   // GBK_TO_UNICODE[27068] := 16#CFB8;
   // GBK_TO_UNICODE[27069] := 16#7EC6;
   // GBK_TO_UNICODE[27070] := 16#CFB9;
   // GBK_TO_UNICODE[27071] := 16#778E;
   // GBK_TO_UNICODE[27072] := 16#CFBA;
   // GBK_TO_UNICODE[27073] := 16#867E;
   // GBK_TO_UNICODE[27074] := 16#CFBB;
   // GBK_TO_UNICODE[27075] := 16#5323;
   // GBK_TO_UNICODE[27076] := 16#CFBC;
   // GBK_TO_UNICODE[27077] := 16#971E;
   // GBK_TO_UNICODE[27078] := 16#CFBD;
   // GBK_TO_UNICODE[27079] := 16#8F96;
   // GBK_TO_UNICODE[27080] := 16#CFBE;
   // GBK_TO_UNICODE[27081] := 16#6687;
   // GBK_TO_UNICODE[27082] := 16#CFBF;
   // GBK_TO_UNICODE[27083] := 16#5CE1;
   // GBK_TO_UNICODE[27084] := 16#CFC0;
   // GBK_TO_UNICODE[27085] := 16#4FA0;
   // GBK_TO_UNICODE[27086] := 16#CFC1;
   // GBK_TO_UNICODE[27087] := 16#72ED;
   // GBK_TO_UNICODE[27088] := 16#CFC2;
   // GBK_TO_UNICODE[27089] := 16#4E0B;
   // GBK_TO_UNICODE[27090] := 16#CFC3;
   // GBK_TO_UNICODE[27091] := 16#53A6;
   // GBK_TO_UNICODE[27092] := 16#CFC4;
   // GBK_TO_UNICODE[27093] := 16#590F;
   // GBK_TO_UNICODE[27094] := 16#CFC5;
   // GBK_TO_UNICODE[27095] := 16#5413;
   // GBK_TO_UNICODE[27096] := 16#CFC6;
   // GBK_TO_UNICODE[27097] := 16#6380;
   // GBK_TO_UNICODE[27098] := 16#CFC7;
   // GBK_TO_UNICODE[27099] := 16#9528;
   // GBK_TO_UNICODE[27100] := 16#CFC8;
   // GBK_TO_UNICODE[27101] := 16#5148;
   // GBK_TO_UNICODE[27102] := 16#CFC9;
   // GBK_TO_UNICODE[27103] := 16#4ED9;
   // GBK_TO_UNICODE[27104] := 16#CFCA;
   // GBK_TO_UNICODE[27105] := 16#9C9C;
   // GBK_TO_UNICODE[27106] := 16#CFCB;
   // GBK_TO_UNICODE[27107] := 16#7EA4;
   // GBK_TO_UNICODE[27108] := 16#CFCC;
   // GBK_TO_UNICODE[27109] := 16#54B8;
   // GBK_TO_UNICODE[27110] := 16#CFCD;
   // GBK_TO_UNICODE[27111] := 16#8D24;
   // GBK_TO_UNICODE[27112] := 16#CFCE;
   // GBK_TO_UNICODE[27113] := 16#8854;
   // GBK_TO_UNICODE[27114] := 16#CFCF;
   // GBK_TO_UNICODE[27115] := 16#8237;
   // GBK_TO_UNICODE[27116] := 16#CFD0;
   // GBK_TO_UNICODE[27117] := 16#95F2;
   // GBK_TO_UNICODE[27118] := 16#CFD1;
   // GBK_TO_UNICODE[27119] := 16#6D8E;
   // GBK_TO_UNICODE[27120] := 16#CFD2;
   // GBK_TO_UNICODE[27121] := 16#5F26;
   // GBK_TO_UNICODE[27122] := 16#CFD3;
   // GBK_TO_UNICODE[27123] := 16#5ACC;
   // GBK_TO_UNICODE[27124] := 16#CFD4;
   // GBK_TO_UNICODE[27125] := 16#663E;
   // GBK_TO_UNICODE[27126] := 16#CFD5;
   // GBK_TO_UNICODE[27127] := 16#9669;
   // GBK_TO_UNICODE[27128] := 16#CFD6;
   // GBK_TO_UNICODE[27129] := 16#73B0;
   // GBK_TO_UNICODE[27130] := 16#CFD7;
   // GBK_TO_UNICODE[27131] := 16#732E;
   // GBK_TO_UNICODE[27132] := 16#CFD8;
   // GBK_TO_UNICODE[27133] := 16#53BF;
   // GBK_TO_UNICODE[27134] := 16#CFD9;
   // GBK_TO_UNICODE[27135] := 16#817A;
   // GBK_TO_UNICODE[27136] := 16#CFDA;
   // GBK_TO_UNICODE[27137] := 16#9985;
   // GBK_TO_UNICODE[27138] := 16#CFDB;
   // GBK_TO_UNICODE[27139] := 16#7FA1;
   // GBK_TO_UNICODE[27140] := 16#CFDC;
   // GBK_TO_UNICODE[27141] := 16#5BAA;
   // GBK_TO_UNICODE[27142] := 16#CFDD;
   // GBK_TO_UNICODE[27143] := 16#9677;
   // GBK_TO_UNICODE[27144] := 16#CFDE;
   // GBK_TO_UNICODE[27145] := 16#9650;
   // GBK_TO_UNICODE[27146] := 16#CFDF;
   // GBK_TO_UNICODE[27147] := 16#7EBF;
   // GBK_TO_UNICODE[27148] := 16#CFE0;
   // GBK_TO_UNICODE[27149] := 16#76F8;
   // GBK_TO_UNICODE[27150] := 16#CFE1;
   // GBK_TO_UNICODE[27151] := 16#53A2;
   // GBK_TO_UNICODE[27152] := 16#CFE2;
   // GBK_TO_UNICODE[27153] := 16#9576;
   // GBK_TO_UNICODE[27154] := 16#CFE3;
   // GBK_TO_UNICODE[27155] := 16#9999;
   // GBK_TO_UNICODE[27156] := 16#CFE4;
   // GBK_TO_UNICODE[27157] := 16#7BB1;
   // GBK_TO_UNICODE[27158] := 16#CFE5;
   // GBK_TO_UNICODE[27159] := 16#8944;
   // GBK_TO_UNICODE[27160] := 16#CFE6;
   // GBK_TO_UNICODE[27161] := 16#6E58;
   // GBK_TO_UNICODE[27162] := 16#CFE7;
   // GBK_TO_UNICODE[27163] := 16#4E61;
   // GBK_TO_UNICODE[27164] := 16#CFE8;
   // GBK_TO_UNICODE[27165] := 16#7FD4;
   // GBK_TO_UNICODE[27166] := 16#CFE9;
   // GBK_TO_UNICODE[27167] := 16#7965;
   // GBK_TO_UNICODE[27168] := 16#CFEA;
   // GBK_TO_UNICODE[27169] := 16#8BE6;
   // GBK_TO_UNICODE[27170] := 16#CFEB;
   // GBK_TO_UNICODE[27171] := 16#60F3;
   // GBK_TO_UNICODE[27172] := 16#CFEC;
   // GBK_TO_UNICODE[27173] := 16#54CD;
   // GBK_TO_UNICODE[27174] := 16#CFED;
   // GBK_TO_UNICODE[27175] := 16#4EAB;
   // GBK_TO_UNICODE[27176] := 16#CFEE;
   // GBK_TO_UNICODE[27177] := 16#9879;
   // GBK_TO_UNICODE[27178] := 16#CFEF;
   // GBK_TO_UNICODE[27179] := 16#5DF7;
   // GBK_TO_UNICODE[27180] := 16#CFF0;
   // GBK_TO_UNICODE[27181] := 16#6A61;
   // GBK_TO_UNICODE[27182] := 16#CFF1;
   // GBK_TO_UNICODE[27183] := 16#50CF;
   // GBK_TO_UNICODE[27184] := 16#CFF2;
   // GBK_TO_UNICODE[27185] := 16#5411;
   // GBK_TO_UNICODE[27186] := 16#CFF3;
   // GBK_TO_UNICODE[27187] := 16#8C61;
   // GBK_TO_UNICODE[27188] := 16#CFF4;
   // GBK_TO_UNICODE[27189] := 16#8427;
   // GBK_TO_UNICODE[27190] := 16#CFF5;
   // GBK_TO_UNICODE[27191] := 16#785D;
   // GBK_TO_UNICODE[27192] := 16#CFF6;
   // GBK_TO_UNICODE[27193] := 16#9704;
   // GBK_TO_UNICODE[27194] := 16#CFF7;
   // GBK_TO_UNICODE[27195] := 16#524A;
   // GBK_TO_UNICODE[27196] := 16#CFF8;
   // GBK_TO_UNICODE[27197] := 16#54EE;
   // GBK_TO_UNICODE[27198] := 16#CFF9;
   // GBK_TO_UNICODE[27199] := 16#56A3;
   // GBK_TO_UNICODE[27200] := 16#CFFA;
   // GBK_TO_UNICODE[27201] := 16#9500;
   // GBK_TO_UNICODE[27202] := 16#CFFB;
   // GBK_TO_UNICODE[27203] := 16#6D88;
   // GBK_TO_UNICODE[27204] := 16#CFFC;
   // GBK_TO_UNICODE[27205] := 16#5BB5;
   // GBK_TO_UNICODE[27206] := 16#CFFD;
   // GBK_TO_UNICODE[27207] := 16#6DC6;
   // GBK_TO_UNICODE[27208] := 16#CFFE;
   // GBK_TO_UNICODE[27209] := 16#6653;
   // GBK_TO_UNICODE[27210] := 16#D040;
   // GBK_TO_UNICODE[27211] := 16#8824;
   // GBK_TO_UNICODE[27212] := 16#D041;
   // GBK_TO_UNICODE[27213] := 16#8825;
   // GBK_TO_UNICODE[27214] := 16#D042;
   // GBK_TO_UNICODE[27215] := 16#8826;
   // GBK_TO_UNICODE[27216] := 16#D043;
   // GBK_TO_UNICODE[27217] := 16#8827;
   // GBK_TO_UNICODE[27218] := 16#D044;
   // GBK_TO_UNICODE[27219] := 16#8828;
   // GBK_TO_UNICODE[27220] := 16#D045;
   // GBK_TO_UNICODE[27221] := 16#8829;
   // GBK_TO_UNICODE[27222] := 16#D046;
   // GBK_TO_UNICODE[27223] := 16#882A;
   // GBK_TO_UNICODE[27224] := 16#D047;
   // GBK_TO_UNICODE[27225] := 16#882B;
   // GBK_TO_UNICODE[27226] := 16#D048;
   // GBK_TO_UNICODE[27227] := 16#882C;
   // GBK_TO_UNICODE[27228] := 16#D049;
   // GBK_TO_UNICODE[27229] := 16#882D;
   // GBK_TO_UNICODE[27230] := 16#D04A;
   // GBK_TO_UNICODE[27231] := 16#882E;
   // GBK_TO_UNICODE[27232] := 16#D04B;
   // GBK_TO_UNICODE[27233] := 16#882F;
   // GBK_TO_UNICODE[27234] := 16#D04C;
   // GBK_TO_UNICODE[27235] := 16#8830;
   // GBK_TO_UNICODE[27236] := 16#D04D;
   // GBK_TO_UNICODE[27237] := 16#8831;
   // GBK_TO_UNICODE[27238] := 16#D04E;
   // GBK_TO_UNICODE[27239] := 16#8833;
   // GBK_TO_UNICODE[27240] := 16#D04F;
   // GBK_TO_UNICODE[27241] := 16#8834;
   // GBK_TO_UNICODE[27242] := 16#D050;
   // GBK_TO_UNICODE[27243] := 16#8835;
   // GBK_TO_UNICODE[27244] := 16#D051;
   // GBK_TO_UNICODE[27245] := 16#8836;
   // GBK_TO_UNICODE[27246] := 16#D052;
   // GBK_TO_UNICODE[27247] := 16#8837;
   // GBK_TO_UNICODE[27248] := 16#D053;
   // GBK_TO_UNICODE[27249] := 16#8838;
   // GBK_TO_UNICODE[27250] := 16#D054;
   // GBK_TO_UNICODE[27251] := 16#883A;
   // GBK_TO_UNICODE[27252] := 16#D055;
   // GBK_TO_UNICODE[27253] := 16#883B;
   // GBK_TO_UNICODE[27254] := 16#D056;
   // GBK_TO_UNICODE[27255] := 16#883D;
   // GBK_TO_UNICODE[27256] := 16#D057;
   // GBK_TO_UNICODE[27257] := 16#883E;
   // GBK_TO_UNICODE[27258] := 16#D058;
   // GBK_TO_UNICODE[27259] := 16#883F;
   // GBK_TO_UNICODE[27260] := 16#D059;
   // GBK_TO_UNICODE[27261] := 16#8841;
   // GBK_TO_UNICODE[27262] := 16#D05A;
   // GBK_TO_UNICODE[27263] := 16#8842;
   // GBK_TO_UNICODE[27264] := 16#D05B;
   // GBK_TO_UNICODE[27265] := 16#8843;
   // GBK_TO_UNICODE[27266] := 16#D05C;
   // GBK_TO_UNICODE[27267] := 16#8846;
   // GBK_TO_UNICODE[27268] := 16#D05D;
   // GBK_TO_UNICODE[27269] := 16#8847;
   // GBK_TO_UNICODE[27270] := 16#D05E;
   // GBK_TO_UNICODE[27271] := 16#8848;
   // GBK_TO_UNICODE[27272] := 16#D05F;
   // GBK_TO_UNICODE[27273] := 16#8849;
   // GBK_TO_UNICODE[27274] := 16#D060;
   // GBK_TO_UNICODE[27275] := 16#884A;
   // GBK_TO_UNICODE[27276] := 16#D061;
   // GBK_TO_UNICODE[27277] := 16#884B;
   // GBK_TO_UNICODE[27278] := 16#D062;
   // GBK_TO_UNICODE[27279] := 16#884E;
   // GBK_TO_UNICODE[27280] := 16#D063;
   // GBK_TO_UNICODE[27281] := 16#884F;
   // GBK_TO_UNICODE[27282] := 16#D064;
   // GBK_TO_UNICODE[27283] := 16#8850;
   // GBK_TO_UNICODE[27284] := 16#D065;
   // GBK_TO_UNICODE[27285] := 16#8851;
   // GBK_TO_UNICODE[27286] := 16#D066;
   // GBK_TO_UNICODE[27287] := 16#8852;
   // GBK_TO_UNICODE[27288] := 16#D067;
   // GBK_TO_UNICODE[27289] := 16#8853;
   // GBK_TO_UNICODE[27290] := 16#D068;
   // GBK_TO_UNICODE[27291] := 16#8855;
   // GBK_TO_UNICODE[27292] := 16#D069;
   // GBK_TO_UNICODE[27293] := 16#8856;
   // GBK_TO_UNICODE[27294] := 16#D06A;
   // GBK_TO_UNICODE[27295] := 16#8858;
   // GBK_TO_UNICODE[27296] := 16#D06B;
   // GBK_TO_UNICODE[27297] := 16#885A;
   // GBK_TO_UNICODE[27298] := 16#D06C;
   // GBK_TO_UNICODE[27299] := 16#885B;
   // GBK_TO_UNICODE[27300] := 16#D06D;
   // GBK_TO_UNICODE[27301] := 16#885C;
   // GBK_TO_UNICODE[27302] := 16#D06E;
   // GBK_TO_UNICODE[27303] := 16#885D;
   // GBK_TO_UNICODE[27304] := 16#D06F;
   // GBK_TO_UNICODE[27305] := 16#885E;
   // GBK_TO_UNICODE[27306] := 16#D070;
   // GBK_TO_UNICODE[27307] := 16#885F;
   // GBK_TO_UNICODE[27308] := 16#D071;
   // GBK_TO_UNICODE[27309] := 16#8860;
   // GBK_TO_UNICODE[27310] := 16#D072;
   // GBK_TO_UNICODE[27311] := 16#8866;
   // GBK_TO_UNICODE[27312] := 16#D073;
   // GBK_TO_UNICODE[27313] := 16#8867;
   // GBK_TO_UNICODE[27314] := 16#D074;
   // GBK_TO_UNICODE[27315] := 16#886A;
   // GBK_TO_UNICODE[27316] := 16#D075;
   // GBK_TO_UNICODE[27317] := 16#886D;
   // GBK_TO_UNICODE[27318] := 16#D076;
   // GBK_TO_UNICODE[27319] := 16#886F;
   // GBK_TO_UNICODE[27320] := 16#D077;
   // GBK_TO_UNICODE[27321] := 16#8871;
   // GBK_TO_UNICODE[27322] := 16#D078;
   // GBK_TO_UNICODE[27323] := 16#8873;
   // GBK_TO_UNICODE[27324] := 16#D079;
   // GBK_TO_UNICODE[27325] := 16#8874;
   // GBK_TO_UNICODE[27326] := 16#D07A;
   // GBK_TO_UNICODE[27327] := 16#8875;
   // GBK_TO_UNICODE[27328] := 16#D07B;
   // GBK_TO_UNICODE[27329] := 16#8876;
   // GBK_TO_UNICODE[27330] := 16#D07C;
   // GBK_TO_UNICODE[27331] := 16#8878;
   // GBK_TO_UNICODE[27332] := 16#D07D;
   // GBK_TO_UNICODE[27333] := 16#8879;
   // GBK_TO_UNICODE[27334] := 16#D07E;
   // GBK_TO_UNICODE[27335] := 16#887A;
   // GBK_TO_UNICODE[27336] := 16#D080;
   // GBK_TO_UNICODE[27337] := 16#887B;
   // GBK_TO_UNICODE[27338] := 16#D081;
   // GBK_TO_UNICODE[27339] := 16#887C;
   // GBK_TO_UNICODE[27340] := 16#D082;
   // GBK_TO_UNICODE[27341] := 16#8880;
   // GBK_TO_UNICODE[27342] := 16#D083;
   // GBK_TO_UNICODE[27343] := 16#8883;
   // GBK_TO_UNICODE[27344] := 16#D084;
   // GBK_TO_UNICODE[27345] := 16#8886;
   // GBK_TO_UNICODE[27346] := 16#D085;
   // GBK_TO_UNICODE[27347] := 16#8887;
   // GBK_TO_UNICODE[27348] := 16#D086;
   // GBK_TO_UNICODE[27349] := 16#8889;
   // GBK_TO_UNICODE[27350] := 16#D087;
   // GBK_TO_UNICODE[27351] := 16#888A;
   // GBK_TO_UNICODE[27352] := 16#D088;
   // GBK_TO_UNICODE[27353] := 16#888C;
   // GBK_TO_UNICODE[27354] := 16#D089;
   // GBK_TO_UNICODE[27355] := 16#888E;
   // GBK_TO_UNICODE[27356] := 16#D08A;
   // GBK_TO_UNICODE[27357] := 16#888F;
   // GBK_TO_UNICODE[27358] := 16#D08B;
   // GBK_TO_UNICODE[27359] := 16#8890;
   // GBK_TO_UNICODE[27360] := 16#D08C;
   // GBK_TO_UNICODE[27361] := 16#8891;
   // GBK_TO_UNICODE[27362] := 16#D08D;
   // GBK_TO_UNICODE[27363] := 16#8893;
   // GBK_TO_UNICODE[27364] := 16#D08E;
   // GBK_TO_UNICODE[27365] := 16#8894;
   // GBK_TO_UNICODE[27366] := 16#D08F;
   // GBK_TO_UNICODE[27367] := 16#8895;
   // GBK_TO_UNICODE[27368] := 16#D090;
   // GBK_TO_UNICODE[27369] := 16#8897;
   // GBK_TO_UNICODE[27370] := 16#D091;
   // GBK_TO_UNICODE[27371] := 16#8898;
   // GBK_TO_UNICODE[27372] := 16#D092;
   // GBK_TO_UNICODE[27373] := 16#8899;
   // GBK_TO_UNICODE[27374] := 16#D093;
   // GBK_TO_UNICODE[27375] := 16#889A;
   // GBK_TO_UNICODE[27376] := 16#D094;
   // GBK_TO_UNICODE[27377] := 16#889B;
   // GBK_TO_UNICODE[27378] := 16#D095;
   // GBK_TO_UNICODE[27379] := 16#889D;
   // GBK_TO_UNICODE[27380] := 16#D096;
   // GBK_TO_UNICODE[27381] := 16#889E;
   // GBK_TO_UNICODE[27382] := 16#D097;
   // GBK_TO_UNICODE[27383] := 16#889F;
   // GBK_TO_UNICODE[27384] := 16#D098;
   // GBK_TO_UNICODE[27385] := 16#88A0;
   // GBK_TO_UNICODE[27386] := 16#D099;
   // GBK_TO_UNICODE[27387] := 16#88A1;
   // GBK_TO_UNICODE[27388] := 16#D09A;
   // GBK_TO_UNICODE[27389] := 16#88A3;
   // GBK_TO_UNICODE[27390] := 16#D09B;
   // GBK_TO_UNICODE[27391] := 16#88A5;
   // GBK_TO_UNICODE[27392] := 16#D09C;
   // GBK_TO_UNICODE[27393] := 16#88A6;
   // GBK_TO_UNICODE[27394] := 16#D09D;
   // GBK_TO_UNICODE[27395] := 16#88A7;
   // GBK_TO_UNICODE[27396] := 16#D09E;
   // GBK_TO_UNICODE[27397] := 16#88A8;
   // GBK_TO_UNICODE[27398] := 16#D09F;
   // GBK_TO_UNICODE[27399] := 16#88A9;
   // GBK_TO_UNICODE[27400] := 16#D0A0;
   // GBK_TO_UNICODE[27401] := 16#88AA;
   // GBK_TO_UNICODE[27402] := 16#D0A1;
   // GBK_TO_UNICODE[27403] := 16#5C0F;
   // GBK_TO_UNICODE[27404] := 16#D0A2;
   // GBK_TO_UNICODE[27405] := 16#5B5D;
   // GBK_TO_UNICODE[27406] := 16#D0A3;
   // GBK_TO_UNICODE[27407] := 16#6821;
   // GBK_TO_UNICODE[27408] := 16#D0A4;
   // GBK_TO_UNICODE[27409] := 16#8096;
   // GBK_TO_UNICODE[27410] := 16#D0A5;
   // GBK_TO_UNICODE[27411] := 16#5578;
   // GBK_TO_UNICODE[27412] := 16#D0A6;
   // GBK_TO_UNICODE[27413] := 16#7B11;
   // GBK_TO_UNICODE[27414] := 16#D0A7;
   // GBK_TO_UNICODE[27415] := 16#6548;
   // GBK_TO_UNICODE[27416] := 16#D0A8;
   // GBK_TO_UNICODE[27417] := 16#6954;
   // GBK_TO_UNICODE[27418] := 16#D0A9;
   // GBK_TO_UNICODE[27419] := 16#4E9B;
   // GBK_TO_UNICODE[27420] := 16#D0AA;
   // GBK_TO_UNICODE[27421] := 16#6B47;
   // GBK_TO_UNICODE[27422] := 16#D0AB;
   // GBK_TO_UNICODE[27423] := 16#874E;
   // GBK_TO_UNICODE[27424] := 16#D0AC;
   // GBK_TO_UNICODE[27425] := 16#978B;
   // GBK_TO_UNICODE[27426] := 16#D0AD;
   // GBK_TO_UNICODE[27427] := 16#534F;
   // GBK_TO_UNICODE[27428] := 16#D0AE;
   // GBK_TO_UNICODE[27429] := 16#631F;
   // GBK_TO_UNICODE[27430] := 16#D0AF;
   // GBK_TO_UNICODE[27431] := 16#643A;
   // GBK_TO_UNICODE[27432] := 16#D0B0;
   // GBK_TO_UNICODE[27433] := 16#90AA;
   // GBK_TO_UNICODE[27434] := 16#D0B1;
   // GBK_TO_UNICODE[27435] := 16#659C;
   // GBK_TO_UNICODE[27436] := 16#D0B2;
   // GBK_TO_UNICODE[27437] := 16#80C1;
   // GBK_TO_UNICODE[27438] := 16#D0B3;
   // GBK_TO_UNICODE[27439] := 16#8C10;
   // GBK_TO_UNICODE[27440] := 16#D0B4;
   // GBK_TO_UNICODE[27441] := 16#5199;
   // GBK_TO_UNICODE[27442] := 16#D0B5;
   // GBK_TO_UNICODE[27443] := 16#68B0;
   // GBK_TO_UNICODE[27444] := 16#D0B6;
   // GBK_TO_UNICODE[27445] := 16#5378;
   // GBK_TO_UNICODE[27446] := 16#D0B7;
   // GBK_TO_UNICODE[27447] := 16#87F9;
   // GBK_TO_UNICODE[27448] := 16#D0B8;
   // GBK_TO_UNICODE[27449] := 16#61C8;
   // GBK_TO_UNICODE[27450] := 16#D0B9;
   // GBK_TO_UNICODE[27451] := 16#6CC4;
   // GBK_TO_UNICODE[27452] := 16#D0BA;
   // GBK_TO_UNICODE[27453] := 16#6CFB;
   // GBK_TO_UNICODE[27454] := 16#D0BB;
   // GBK_TO_UNICODE[27455] := 16#8C22;
   // GBK_TO_UNICODE[27456] := 16#D0BC;
   // GBK_TO_UNICODE[27457] := 16#5C51;
   // GBK_TO_UNICODE[27458] := 16#D0BD;
   // GBK_TO_UNICODE[27459] := 16#85AA;
   // GBK_TO_UNICODE[27460] := 16#D0BE;
   // GBK_TO_UNICODE[27461] := 16#82AF;
   // GBK_TO_UNICODE[27462] := 16#D0BF;
   // GBK_TO_UNICODE[27463] := 16#950C;
   // GBK_TO_UNICODE[27464] := 16#D0C0;
   // GBK_TO_UNICODE[27465] := 16#6B23;
   // GBK_TO_UNICODE[27466] := 16#D0C1;
   // GBK_TO_UNICODE[27467] := 16#8F9B;
   // GBK_TO_UNICODE[27468] := 16#D0C2;
   // GBK_TO_UNICODE[27469] := 16#65B0;
   // GBK_TO_UNICODE[27470] := 16#D0C3;
   // GBK_TO_UNICODE[27471] := 16#5FFB;
   // GBK_TO_UNICODE[27472] := 16#D0C4;
   // GBK_TO_UNICODE[27473] := 16#5FC3;
   // GBK_TO_UNICODE[27474] := 16#D0C5;
   // GBK_TO_UNICODE[27475] := 16#4FE1;
   // GBK_TO_UNICODE[27476] := 16#D0C6;
   // GBK_TO_UNICODE[27477] := 16#8845;
   // GBK_TO_UNICODE[27478] := 16#D0C7;
   // GBK_TO_UNICODE[27479] := 16#661F;
   // GBK_TO_UNICODE[27480] := 16#D0C8;
   // GBK_TO_UNICODE[27481] := 16#8165;
   // GBK_TO_UNICODE[27482] := 16#D0C9;
   // GBK_TO_UNICODE[27483] := 16#7329;
   // GBK_TO_UNICODE[27484] := 16#D0CA;
   // GBK_TO_UNICODE[27485] := 16#60FA;
   // GBK_TO_UNICODE[27486] := 16#D0CB;
   // GBK_TO_UNICODE[27487] := 16#5174;
   // GBK_TO_UNICODE[27488] := 16#D0CC;
   // GBK_TO_UNICODE[27489] := 16#5211;
   // GBK_TO_UNICODE[27490] := 16#D0CD;
   // GBK_TO_UNICODE[27491] := 16#578B;
   // GBK_TO_UNICODE[27492] := 16#D0CE;
   // GBK_TO_UNICODE[27493] := 16#5F62;
   // GBK_TO_UNICODE[27494] := 16#D0CF;
   // GBK_TO_UNICODE[27495] := 16#90A2;
   // GBK_TO_UNICODE[27496] := 16#D0D0;
   // GBK_TO_UNICODE[27497] := 16#884C;
   // GBK_TO_UNICODE[27498] := 16#D0D1;
   // GBK_TO_UNICODE[27499] := 16#9192;
   // GBK_TO_UNICODE[27500] := 16#D0D2;
   // GBK_TO_UNICODE[27501] := 16#5E78;
   // GBK_TO_UNICODE[27502] := 16#D0D3;
   // GBK_TO_UNICODE[27503] := 16#674F;
   // GBK_TO_UNICODE[27504] := 16#D0D4;
   // GBK_TO_UNICODE[27505] := 16#6027;
   // GBK_TO_UNICODE[27506] := 16#D0D5;
   // GBK_TO_UNICODE[27507] := 16#59D3;
   // GBK_TO_UNICODE[27508] := 16#D0D6;
   // GBK_TO_UNICODE[27509] := 16#5144;
   // GBK_TO_UNICODE[27510] := 16#D0D7;
   // GBK_TO_UNICODE[27511] := 16#51F6;
   // GBK_TO_UNICODE[27512] := 16#D0D8;
   // GBK_TO_UNICODE[27513] := 16#80F8;
   // GBK_TO_UNICODE[27514] := 16#D0D9;
   // GBK_TO_UNICODE[27515] := 16#5308;
   // GBK_TO_UNICODE[27516] := 16#D0DA;
   // GBK_TO_UNICODE[27517] := 16#6C79;
   // GBK_TO_UNICODE[27518] := 16#D0DB;
   // GBK_TO_UNICODE[27519] := 16#96C4;
   // GBK_TO_UNICODE[27520] := 16#D0DC;
   // GBK_TO_UNICODE[27521] := 16#718A;
   // GBK_TO_UNICODE[27522] := 16#D0DD;
   // GBK_TO_UNICODE[27523] := 16#4F11;
   // GBK_TO_UNICODE[27524] := 16#D0DE;
   // GBK_TO_UNICODE[27525] := 16#4FEE;
   // GBK_TO_UNICODE[27526] := 16#D0DF;
   // GBK_TO_UNICODE[27527] := 16#7F9E;
   // GBK_TO_UNICODE[27528] := 16#D0E0;
   // GBK_TO_UNICODE[27529] := 16#673D;
   // GBK_TO_UNICODE[27530] := 16#D0E1;
   // GBK_TO_UNICODE[27531] := 16#55C5;
   // GBK_TO_UNICODE[27532] := 16#D0E2;
   // GBK_TO_UNICODE[27533] := 16#9508;
   // GBK_TO_UNICODE[27534] := 16#D0E3;
   // GBK_TO_UNICODE[27535] := 16#79C0;
   // GBK_TO_UNICODE[27536] := 16#D0E4;
   // GBK_TO_UNICODE[27537] := 16#8896;
   // GBK_TO_UNICODE[27538] := 16#D0E5;
   // GBK_TO_UNICODE[27539] := 16#7EE3;
   // GBK_TO_UNICODE[27540] := 16#D0E6;
   // GBK_TO_UNICODE[27541] := 16#589F;
   // GBK_TO_UNICODE[27542] := 16#D0E7;
   // GBK_TO_UNICODE[27543] := 16#620C;
   // GBK_TO_UNICODE[27544] := 16#D0E8;
   // GBK_TO_UNICODE[27545] := 16#9700;
   // GBK_TO_UNICODE[27546] := 16#D0E9;
   // GBK_TO_UNICODE[27547] := 16#865A;
   // GBK_TO_UNICODE[27548] := 16#D0EA;
   // GBK_TO_UNICODE[27549] := 16#5618;
   // GBK_TO_UNICODE[27550] := 16#D0EB;
   // GBK_TO_UNICODE[27551] := 16#987B;
   // GBK_TO_UNICODE[27552] := 16#D0EC;
   // GBK_TO_UNICODE[27553] := 16#5F90;
   // GBK_TO_UNICODE[27554] := 16#D0ED;
   // GBK_TO_UNICODE[27555] := 16#8BB8;
   // GBK_TO_UNICODE[27556] := 16#D0EE;
   // GBK_TO_UNICODE[27557] := 16#84C4;
   // GBK_TO_UNICODE[27558] := 16#D0EF;
   // GBK_TO_UNICODE[27559] := 16#9157;
   // GBK_TO_UNICODE[27560] := 16#D0F0;
   // GBK_TO_UNICODE[27561] := 16#53D9;
   // GBK_TO_UNICODE[27562] := 16#D0F1;
   // GBK_TO_UNICODE[27563] := 16#65ED;
   // GBK_TO_UNICODE[27564] := 16#D0F2;
   // GBK_TO_UNICODE[27565] := 16#5E8F;
   // GBK_TO_UNICODE[27566] := 16#D0F3;
   // GBK_TO_UNICODE[27567] := 16#755C;
   // GBK_TO_UNICODE[27568] := 16#D0F4;
   // GBK_TO_UNICODE[27569] := 16#6064;
   // GBK_TO_UNICODE[27570] := 16#D0F5;
   // GBK_TO_UNICODE[27571] := 16#7D6E;
   // GBK_TO_UNICODE[27572] := 16#D0F6;
   // GBK_TO_UNICODE[27573] := 16#5A7F;
   // GBK_TO_UNICODE[27574] := 16#D0F7;
   // GBK_TO_UNICODE[27575] := 16#7EEA;
   // GBK_TO_UNICODE[27576] := 16#D0F8;
   // GBK_TO_UNICODE[27577] := 16#7EED;
   // GBK_TO_UNICODE[27578] := 16#D0F9;
   // GBK_TO_UNICODE[27579] := 16#8F69;
   // GBK_TO_UNICODE[27580] := 16#D0FA;
   // GBK_TO_UNICODE[27581] := 16#55A7;
   // GBK_TO_UNICODE[27582] := 16#D0FB;
   // GBK_TO_UNICODE[27583] := 16#5BA3;
   // GBK_TO_UNICODE[27584] := 16#D0FC;
   // GBK_TO_UNICODE[27585] := 16#60AC;
   // GBK_TO_UNICODE[27586] := 16#D0FD;
   // GBK_TO_UNICODE[27587] := 16#65CB;
   // GBK_TO_UNICODE[27588] := 16#D0FE;
   // GBK_TO_UNICODE[27589] := 16#7384;
   // GBK_TO_UNICODE[27590] := 16#D140;
   // GBK_TO_UNICODE[27591] := 16#88AC;
   // GBK_TO_UNICODE[27592] := 16#D141;
   // GBK_TO_UNICODE[27593] := 16#88AE;
   // GBK_TO_UNICODE[27594] := 16#D142;
   // GBK_TO_UNICODE[27595] := 16#88AF;
   // GBK_TO_UNICODE[27596] := 16#D143;
   // GBK_TO_UNICODE[27597] := 16#88B0;
   // GBK_TO_UNICODE[27598] := 16#D144;
   // GBK_TO_UNICODE[27599] := 16#88B2;
   // GBK_TO_UNICODE[27600] := 16#D145;
   // GBK_TO_UNICODE[27601] := 16#88B3;
   // GBK_TO_UNICODE[27602] := 16#D146;
   // GBK_TO_UNICODE[27603] := 16#88B4;
   // GBK_TO_UNICODE[27604] := 16#D147;
   // GBK_TO_UNICODE[27605] := 16#88B5;
   // GBK_TO_UNICODE[27606] := 16#D148;
   // GBK_TO_UNICODE[27607] := 16#88B6;
   // GBK_TO_UNICODE[27608] := 16#D149;
   // GBK_TO_UNICODE[27609] := 16#88B8;
   // GBK_TO_UNICODE[27610] := 16#D14A;
   // GBK_TO_UNICODE[27611] := 16#88B9;
   // GBK_TO_UNICODE[27612] := 16#D14B;
   // GBK_TO_UNICODE[27613] := 16#88BA;
   // GBK_TO_UNICODE[27614] := 16#D14C;
   // GBK_TO_UNICODE[27615] := 16#88BB;
   // GBK_TO_UNICODE[27616] := 16#D14D;
   // GBK_TO_UNICODE[27617] := 16#88BD;
   // GBK_TO_UNICODE[27618] := 16#D14E;
   // GBK_TO_UNICODE[27619] := 16#88BE;
   // GBK_TO_UNICODE[27620] := 16#D14F;
   // GBK_TO_UNICODE[27621] := 16#88BF;
   // GBK_TO_UNICODE[27622] := 16#D150;
   // GBK_TO_UNICODE[27623] := 16#88C0;
   // GBK_TO_UNICODE[27624] := 16#D151;
   // GBK_TO_UNICODE[27625] := 16#88C3;
   // GBK_TO_UNICODE[27626] := 16#D152;
   // GBK_TO_UNICODE[27627] := 16#88C4;
   // GBK_TO_UNICODE[27628] := 16#D153;
   // GBK_TO_UNICODE[27629] := 16#88C7;
   // GBK_TO_UNICODE[27630] := 16#D154;
   // GBK_TO_UNICODE[27631] := 16#88C8;
   // GBK_TO_UNICODE[27632] := 16#D155;
   // GBK_TO_UNICODE[27633] := 16#88CA;
   // GBK_TO_UNICODE[27634] := 16#D156;
   // GBK_TO_UNICODE[27635] := 16#88CB;
   // GBK_TO_UNICODE[27636] := 16#D157;
   // GBK_TO_UNICODE[27637] := 16#88CC;
   // GBK_TO_UNICODE[27638] := 16#D158;
   // GBK_TO_UNICODE[27639] := 16#88CD;
   // GBK_TO_UNICODE[27640] := 16#D159;
   // GBK_TO_UNICODE[27641] := 16#88CF;
   // GBK_TO_UNICODE[27642] := 16#D15A;
   // GBK_TO_UNICODE[27643] := 16#88D0;
   // GBK_TO_UNICODE[27644] := 16#D15B;
   // GBK_TO_UNICODE[27645] := 16#88D1;
   // GBK_TO_UNICODE[27646] := 16#D15C;
   // GBK_TO_UNICODE[27647] := 16#88D3;
   // GBK_TO_UNICODE[27648] := 16#D15D;
   // GBK_TO_UNICODE[27649] := 16#88D6;
   // GBK_TO_UNICODE[27650] := 16#D15E;
   // GBK_TO_UNICODE[27651] := 16#88D7;
   // GBK_TO_UNICODE[27652] := 16#D15F;
   // GBK_TO_UNICODE[27653] := 16#88DA;
   // GBK_TO_UNICODE[27654] := 16#D160;
   // GBK_TO_UNICODE[27655] := 16#88DB;
   // GBK_TO_UNICODE[27656] := 16#D161;
   // GBK_TO_UNICODE[27657] := 16#88DC;
   // GBK_TO_UNICODE[27658] := 16#D162;
   // GBK_TO_UNICODE[27659] := 16#88DD;
   // GBK_TO_UNICODE[27660] := 16#D163;
   // GBK_TO_UNICODE[27661] := 16#88DE;
   // GBK_TO_UNICODE[27662] := 16#D164;
   // GBK_TO_UNICODE[27663] := 16#88E0;
   // GBK_TO_UNICODE[27664] := 16#D165;
   // GBK_TO_UNICODE[27665] := 16#88E1;
   // GBK_TO_UNICODE[27666] := 16#D166;
   // GBK_TO_UNICODE[27667] := 16#88E6;
   // GBK_TO_UNICODE[27668] := 16#D167;
   // GBK_TO_UNICODE[27669] := 16#88E7;
   // GBK_TO_UNICODE[27670] := 16#D168;
   // GBK_TO_UNICODE[27671] := 16#88E9;
   // GBK_TO_UNICODE[27672] := 16#D169;
   // GBK_TO_UNICODE[27673] := 16#88EA;
   // GBK_TO_UNICODE[27674] := 16#D16A;
   // GBK_TO_UNICODE[27675] := 16#88EB;
   // GBK_TO_UNICODE[27676] := 16#D16B;
   // GBK_TO_UNICODE[27677] := 16#88EC;
   // GBK_TO_UNICODE[27678] := 16#D16C;
   // GBK_TO_UNICODE[27679] := 16#88ED;
   // GBK_TO_UNICODE[27680] := 16#D16D;
   // GBK_TO_UNICODE[27681] := 16#88EE;
   // GBK_TO_UNICODE[27682] := 16#D16E;
   // GBK_TO_UNICODE[27683] := 16#88EF;
   // GBK_TO_UNICODE[27684] := 16#D16F;
   // GBK_TO_UNICODE[27685] := 16#88F2;
   // GBK_TO_UNICODE[27686] := 16#D170;
   // GBK_TO_UNICODE[27687] := 16#88F5;
   // GBK_TO_UNICODE[27688] := 16#D171;
   // GBK_TO_UNICODE[27689] := 16#88F6;
   // GBK_TO_UNICODE[27690] := 16#D172;
   // GBK_TO_UNICODE[27691] := 16#88F7;
   // GBK_TO_UNICODE[27692] := 16#D173;
   // GBK_TO_UNICODE[27693] := 16#88FA;
   // GBK_TO_UNICODE[27694] := 16#D174;
   // GBK_TO_UNICODE[27695] := 16#88FB;
   // GBK_TO_UNICODE[27696] := 16#D175;
   // GBK_TO_UNICODE[27697] := 16#88FD;
   // GBK_TO_UNICODE[27698] := 16#D176;
   // GBK_TO_UNICODE[27699] := 16#88FF;
   // GBK_TO_UNICODE[27700] := 16#D177;
   // GBK_TO_UNICODE[27701] := 16#8900;
   // GBK_TO_UNICODE[27702] := 16#D178;
   // GBK_TO_UNICODE[27703] := 16#8901;
   // GBK_TO_UNICODE[27704] := 16#D179;
   // GBK_TO_UNICODE[27705] := 16#8903;
   // GBK_TO_UNICODE[27706] := 16#D17A;
   // GBK_TO_UNICODE[27707] := 16#8904;
   // GBK_TO_UNICODE[27708] := 16#D17B;
   // GBK_TO_UNICODE[27709] := 16#8905;
   // GBK_TO_UNICODE[27710] := 16#D17C;
   // GBK_TO_UNICODE[27711] := 16#8906;
   // GBK_TO_UNICODE[27712] := 16#D17D;
   // GBK_TO_UNICODE[27713] := 16#8907;
   // GBK_TO_UNICODE[27714] := 16#D17E;
   // GBK_TO_UNICODE[27715] := 16#8908;
   // GBK_TO_UNICODE[27716] := 16#D180;
   // GBK_TO_UNICODE[27717] := 16#8909;
   // GBK_TO_UNICODE[27718] := 16#D181;
   // GBK_TO_UNICODE[27719] := 16#890B;
   // GBK_TO_UNICODE[27720] := 16#D182;
   // GBK_TO_UNICODE[27721] := 16#890C;
   // GBK_TO_UNICODE[27722] := 16#D183;
   // GBK_TO_UNICODE[27723] := 16#890D;
   // GBK_TO_UNICODE[27724] := 16#D184;
   // GBK_TO_UNICODE[27725] := 16#890E;
   // GBK_TO_UNICODE[27726] := 16#D185;
   // GBK_TO_UNICODE[27727] := 16#890F;
   // GBK_TO_UNICODE[27728] := 16#D186;
   // GBK_TO_UNICODE[27729] := 16#8911;
   // GBK_TO_UNICODE[27730] := 16#D187;
   // GBK_TO_UNICODE[27731] := 16#8914;
   // GBK_TO_UNICODE[27732] := 16#D188;
   // GBK_TO_UNICODE[27733] := 16#8915;
   // GBK_TO_UNICODE[27734] := 16#D189;
   // GBK_TO_UNICODE[27735] := 16#8916;
   // GBK_TO_UNICODE[27736] := 16#D18A;
   // GBK_TO_UNICODE[27737] := 16#8917;
   // GBK_TO_UNICODE[27738] := 16#D18B;
   // GBK_TO_UNICODE[27739] := 16#8918;
   // GBK_TO_UNICODE[27740] := 16#D18C;
   // GBK_TO_UNICODE[27741] := 16#891C;
   // GBK_TO_UNICODE[27742] := 16#D18D;
   // GBK_TO_UNICODE[27743] := 16#891D;
   // GBK_TO_UNICODE[27744] := 16#D18E;
   // GBK_TO_UNICODE[27745] := 16#891E;
   // GBK_TO_UNICODE[27746] := 16#D18F;
   // GBK_TO_UNICODE[27747] := 16#891F;
   // GBK_TO_UNICODE[27748] := 16#D190;
   // GBK_TO_UNICODE[27749] := 16#8920;
   // GBK_TO_UNICODE[27750] := 16#D191;
   // GBK_TO_UNICODE[27751] := 16#8922;
   // GBK_TO_UNICODE[27752] := 16#D192;
   // GBK_TO_UNICODE[27753] := 16#8923;
   // GBK_TO_UNICODE[27754] := 16#D193;
   // GBK_TO_UNICODE[27755] := 16#8924;
   // GBK_TO_UNICODE[27756] := 16#D194;
   // GBK_TO_UNICODE[27757] := 16#8926;
   // GBK_TO_UNICODE[27758] := 16#D195;
   // GBK_TO_UNICODE[27759] := 16#8927;
   // GBK_TO_UNICODE[27760] := 16#D196;
   // GBK_TO_UNICODE[27761] := 16#8928;
   // GBK_TO_UNICODE[27762] := 16#D197;
   // GBK_TO_UNICODE[27763] := 16#8929;
   // GBK_TO_UNICODE[27764] := 16#D198;
   // GBK_TO_UNICODE[27765] := 16#892C;
   // GBK_TO_UNICODE[27766] := 16#D199;
   // GBK_TO_UNICODE[27767] := 16#892D;
   // GBK_TO_UNICODE[27768] := 16#D19A;
   // GBK_TO_UNICODE[27769] := 16#892E;
   // GBK_TO_UNICODE[27770] := 16#D19B;
   // GBK_TO_UNICODE[27771] := 16#892F;
   // GBK_TO_UNICODE[27772] := 16#D19C;
   // GBK_TO_UNICODE[27773] := 16#8931;
   // GBK_TO_UNICODE[27774] := 16#D19D;
   // GBK_TO_UNICODE[27775] := 16#8932;
   // GBK_TO_UNICODE[27776] := 16#D19E;
   // GBK_TO_UNICODE[27777] := 16#8933;
   // GBK_TO_UNICODE[27778] := 16#D19F;
   // GBK_TO_UNICODE[27779] := 16#8935;
   // GBK_TO_UNICODE[27780] := 16#D1A0;
   // GBK_TO_UNICODE[27781] := 16#8937;
   // GBK_TO_UNICODE[27782] := 16#D1A1;
   // GBK_TO_UNICODE[27783] := 16#9009;
   // GBK_TO_UNICODE[27784] := 16#D1A2;
   // GBK_TO_UNICODE[27785] := 16#7663;
   // GBK_TO_UNICODE[27786] := 16#D1A3;
   // GBK_TO_UNICODE[27787] := 16#7729;
   // GBK_TO_UNICODE[27788] := 16#D1A4;
   // GBK_TO_UNICODE[27789] := 16#7EDA;
   // GBK_TO_UNICODE[27790] := 16#D1A5;
   // GBK_TO_UNICODE[27791] := 16#9774;
   // GBK_TO_UNICODE[27792] := 16#D1A6;
   // GBK_TO_UNICODE[27793] := 16#859B;
   // GBK_TO_UNICODE[27794] := 16#D1A7;
   // GBK_TO_UNICODE[27795] := 16#5B66;
   // GBK_TO_UNICODE[27796] := 16#D1A8;
   // GBK_TO_UNICODE[27797] := 16#7A74;
   // GBK_TO_UNICODE[27798] := 16#D1A9;
   // GBK_TO_UNICODE[27799] := 16#96EA;
   // GBK_TO_UNICODE[27800] := 16#D1AA;
   // GBK_TO_UNICODE[27801] := 16#8840;
   // GBK_TO_UNICODE[27802] := 16#D1AB;
   // GBK_TO_UNICODE[27803] := 16#52CB;
   // GBK_TO_UNICODE[27804] := 16#D1AC;
   // GBK_TO_UNICODE[27805] := 16#718F;
   // GBK_TO_UNICODE[27806] := 16#D1AD;
   // GBK_TO_UNICODE[27807] := 16#5FAA;
   // GBK_TO_UNICODE[27808] := 16#D1AE;
   // GBK_TO_UNICODE[27809] := 16#65EC;
   // GBK_TO_UNICODE[27810] := 16#D1AF;
   // GBK_TO_UNICODE[27811] := 16#8BE2;
   // GBK_TO_UNICODE[27812] := 16#D1B0;
   // GBK_TO_UNICODE[27813] := 16#5BFB;
   // GBK_TO_UNICODE[27814] := 16#D1B1;
   // GBK_TO_UNICODE[27815] := 16#9A6F;
   // GBK_TO_UNICODE[27816] := 16#D1B2;
   // GBK_TO_UNICODE[27817] := 16#5DE1;
   // GBK_TO_UNICODE[27818] := 16#D1B3;
   // GBK_TO_UNICODE[27819] := 16#6B89;
   // GBK_TO_UNICODE[27820] := 16#D1B4;
   // GBK_TO_UNICODE[27821] := 16#6C5B;
   // GBK_TO_UNICODE[27822] := 16#D1B5;
   // GBK_TO_UNICODE[27823] := 16#8BAD;
   // GBK_TO_UNICODE[27824] := 16#D1B6;
   // GBK_TO_UNICODE[27825] := 16#8BAF;
   // GBK_TO_UNICODE[27826] := 16#D1B7;
   // GBK_TO_UNICODE[27827] := 16#900A;
   // GBK_TO_UNICODE[27828] := 16#D1B8;
   // GBK_TO_UNICODE[27829] := 16#8FC5;
   // GBK_TO_UNICODE[27830] := 16#D1B9;
   // GBK_TO_UNICODE[27831] := 16#538B;
   // GBK_TO_UNICODE[27832] := 16#D1BA;
   // GBK_TO_UNICODE[27833] := 16#62BC;
   // GBK_TO_UNICODE[27834] := 16#D1BB;
   // GBK_TO_UNICODE[27835] := 16#9E26;
   // GBK_TO_UNICODE[27836] := 16#D1BC;
   // GBK_TO_UNICODE[27837] := 16#9E2D;
   // GBK_TO_UNICODE[27838] := 16#D1BD;
   // GBK_TO_UNICODE[27839] := 16#5440;
   // GBK_TO_UNICODE[27840] := 16#D1BE;
   // GBK_TO_UNICODE[27841] := 16#4E2B;
   // GBK_TO_UNICODE[27842] := 16#D1BF;
   // GBK_TO_UNICODE[27843] := 16#82BD;
   // GBK_TO_UNICODE[27844] := 16#D1C0;
   // GBK_TO_UNICODE[27845] := 16#7259;
   // GBK_TO_UNICODE[27846] := 16#D1C1;
   // GBK_TO_UNICODE[27847] := 16#869C;
   // GBK_TO_UNICODE[27848] := 16#D1C2;
   // GBK_TO_UNICODE[27849] := 16#5D16;
   // GBK_TO_UNICODE[27850] := 16#D1C3;
   // GBK_TO_UNICODE[27851] := 16#8859;
   // GBK_TO_UNICODE[27852] := 16#D1C4;
   // GBK_TO_UNICODE[27853] := 16#6DAF;
   // GBK_TO_UNICODE[27854] := 16#D1C5;
   // GBK_TO_UNICODE[27855] := 16#96C5;
   // GBK_TO_UNICODE[27856] := 16#D1C6;
   // GBK_TO_UNICODE[27857] := 16#54D1;
   // GBK_TO_UNICODE[27858] := 16#D1C7;
   // GBK_TO_UNICODE[27859] := 16#4E9A;
   // GBK_TO_UNICODE[27860] := 16#D1C8;
   // GBK_TO_UNICODE[27861] := 16#8BB6;
   // GBK_TO_UNICODE[27862] := 16#D1C9;
   // GBK_TO_UNICODE[27863] := 16#7109;
   // GBK_TO_UNICODE[27864] := 16#D1CA;
   // GBK_TO_UNICODE[27865] := 16#54BD;
   // GBK_TO_UNICODE[27866] := 16#D1CB;
   // GBK_TO_UNICODE[27867] := 16#9609;
   // GBK_TO_UNICODE[27868] := 16#D1CC;
   // GBK_TO_UNICODE[27869] := 16#70DF;
   // GBK_TO_UNICODE[27870] := 16#D1CD;
   // GBK_TO_UNICODE[27871] := 16#6DF9;
   // GBK_TO_UNICODE[27872] := 16#D1CE;
   // GBK_TO_UNICODE[27873] := 16#76D0;
   // GBK_TO_UNICODE[27874] := 16#D1CF;
   // GBK_TO_UNICODE[27875] := 16#4E25;
   // GBK_TO_UNICODE[27876] := 16#D1D0;
   // GBK_TO_UNICODE[27877] := 16#7814;
   // GBK_TO_UNICODE[27878] := 16#D1D1;
   // GBK_TO_UNICODE[27879] := 16#8712;
   // GBK_TO_UNICODE[27880] := 16#D1D2;
   // GBK_TO_UNICODE[27881] := 16#5CA9;
   // GBK_TO_UNICODE[27882] := 16#D1D3;
   // GBK_TO_UNICODE[27883] := 16#5EF6;
   // GBK_TO_UNICODE[27884] := 16#D1D4;
   // GBK_TO_UNICODE[27885] := 16#8A00;
   // GBK_TO_UNICODE[27886] := 16#D1D5;
   // GBK_TO_UNICODE[27887] := 16#989C;
   // GBK_TO_UNICODE[27888] := 16#D1D6;
   // GBK_TO_UNICODE[27889] := 16#960E;
   // GBK_TO_UNICODE[27890] := 16#D1D7;
   // GBK_TO_UNICODE[27891] := 16#708E;
   // GBK_TO_UNICODE[27892] := 16#D1D8;
   // GBK_TO_UNICODE[27893] := 16#6CBF;
   // GBK_TO_UNICODE[27894] := 16#D1D9;
   // GBK_TO_UNICODE[27895] := 16#5944;
   // GBK_TO_UNICODE[27896] := 16#D1DA;
   // GBK_TO_UNICODE[27897] := 16#63A9;
   // GBK_TO_UNICODE[27898] := 16#D1DB;
   // GBK_TO_UNICODE[27899] := 16#773C;
   // GBK_TO_UNICODE[27900] := 16#D1DC;
   // GBK_TO_UNICODE[27901] := 16#884D;
   // GBK_TO_UNICODE[27902] := 16#D1DD;
   // GBK_TO_UNICODE[27903] := 16#6F14;
   // GBK_TO_UNICODE[27904] := 16#D1DE;
   // GBK_TO_UNICODE[27905] := 16#8273;
   // GBK_TO_UNICODE[27906] := 16#D1DF;
   // GBK_TO_UNICODE[27907] := 16#5830;
   // GBK_TO_UNICODE[27908] := 16#D1E0;
   // GBK_TO_UNICODE[27909] := 16#71D5;
   // GBK_TO_UNICODE[27910] := 16#D1E1;
   // GBK_TO_UNICODE[27911] := 16#538C;
   // GBK_TO_UNICODE[27912] := 16#D1E2;
   // GBK_TO_UNICODE[27913] := 16#781A;
   // GBK_TO_UNICODE[27914] := 16#D1E3;
   // GBK_TO_UNICODE[27915] := 16#96C1;
   // GBK_TO_UNICODE[27916] := 16#D1E4;
   // GBK_TO_UNICODE[27917] := 16#5501;
   // GBK_TO_UNICODE[27918] := 16#D1E5;
   // GBK_TO_UNICODE[27919] := 16#5F66;
   // GBK_TO_UNICODE[27920] := 16#D1E6;
   // GBK_TO_UNICODE[27921] := 16#7130;
   // GBK_TO_UNICODE[27922] := 16#D1E7;
   // GBK_TO_UNICODE[27923] := 16#5BB4;
   // GBK_TO_UNICODE[27924] := 16#D1E8;
   // GBK_TO_UNICODE[27925] := 16#8C1A;
   // GBK_TO_UNICODE[27926] := 16#D1E9;
   // GBK_TO_UNICODE[27927] := 16#9A8C;
   // GBK_TO_UNICODE[27928] := 16#D1EA;
   // GBK_TO_UNICODE[27929] := 16#6B83;
   // GBK_TO_UNICODE[27930] := 16#D1EB;
   // GBK_TO_UNICODE[27931] := 16#592E;
   // GBK_TO_UNICODE[27932] := 16#D1EC;
   // GBK_TO_UNICODE[27933] := 16#9E2F;
   // GBK_TO_UNICODE[27934] := 16#D1ED;
   // GBK_TO_UNICODE[27935] := 16#79E7;
   // GBK_TO_UNICODE[27936] := 16#D1EE;
   // GBK_TO_UNICODE[27937] := 16#6768;
   // GBK_TO_UNICODE[27938] := 16#D1EF;
   // GBK_TO_UNICODE[27939] := 16#626C;
   // GBK_TO_UNICODE[27940] := 16#D1F0;
   // GBK_TO_UNICODE[27941] := 16#4F6F;
   // GBK_TO_UNICODE[27942] := 16#D1F1;
   // GBK_TO_UNICODE[27943] := 16#75A1;
   // GBK_TO_UNICODE[27944] := 16#D1F2;
   // GBK_TO_UNICODE[27945] := 16#7F8A;
   // GBK_TO_UNICODE[27946] := 16#D1F3;
   // GBK_TO_UNICODE[27947] := 16#6D0B;
   // GBK_TO_UNICODE[27948] := 16#D1F4;
   // GBK_TO_UNICODE[27949] := 16#9633;
   // GBK_TO_UNICODE[27950] := 16#D1F5;
   // GBK_TO_UNICODE[27951] := 16#6C27;
   // GBK_TO_UNICODE[27952] := 16#D1F6;
   // GBK_TO_UNICODE[27953] := 16#4EF0;
   // GBK_TO_UNICODE[27954] := 16#D1F7;
   // GBK_TO_UNICODE[27955] := 16#75D2;
   // GBK_TO_UNICODE[27956] := 16#D1F8;
   // GBK_TO_UNICODE[27957] := 16#517B;
   // GBK_TO_UNICODE[27958] := 16#D1F9;
   // GBK_TO_UNICODE[27959] := 16#6837;
   // GBK_TO_UNICODE[27960] := 16#D1FA;
   // GBK_TO_UNICODE[27961] := 16#6F3E;
   // GBK_TO_UNICODE[27962] := 16#D1FB;
   // GBK_TO_UNICODE[27963] := 16#9080;
   // GBK_TO_UNICODE[27964] := 16#D1FC;
   // GBK_TO_UNICODE[27965] := 16#8170;
   // GBK_TO_UNICODE[27966] := 16#D1FD;
   // GBK_TO_UNICODE[27967] := 16#5996;
   // GBK_TO_UNICODE[27968] := 16#D1FE;
   // GBK_TO_UNICODE[27969] := 16#7476;
   // GBK_TO_UNICODE[27970] := 16#D240;
   // GBK_TO_UNICODE[27971] := 16#8938;
   // GBK_TO_UNICODE[27972] := 16#D241;
   // GBK_TO_UNICODE[27973] := 16#8939;
   // GBK_TO_UNICODE[27974] := 16#D242;
   // GBK_TO_UNICODE[27975] := 16#893A;
   // GBK_TO_UNICODE[27976] := 16#D243;
   // GBK_TO_UNICODE[27977] := 16#893B;
   // GBK_TO_UNICODE[27978] := 16#D244;
   // GBK_TO_UNICODE[27979] := 16#893C;
   // GBK_TO_UNICODE[27980] := 16#D245;
   // GBK_TO_UNICODE[27981] := 16#893D;
   // GBK_TO_UNICODE[27982] := 16#D246;
   // GBK_TO_UNICODE[27983] := 16#893E;
   // GBK_TO_UNICODE[27984] := 16#D247;
   // GBK_TO_UNICODE[27985] := 16#893F;
   // GBK_TO_UNICODE[27986] := 16#D248;
   // GBK_TO_UNICODE[27987] := 16#8940;
   // GBK_TO_UNICODE[27988] := 16#D249;
   // GBK_TO_UNICODE[27989] := 16#8942;
   // GBK_TO_UNICODE[27990] := 16#D24A;
   // GBK_TO_UNICODE[27991] := 16#8943;
   // GBK_TO_UNICODE[27992] := 16#D24B;
   // GBK_TO_UNICODE[27993] := 16#8945;
   // GBK_TO_UNICODE[27994] := 16#D24C;
   // GBK_TO_UNICODE[27995] := 16#8946;
   // GBK_TO_UNICODE[27996] := 16#D24D;
   // GBK_TO_UNICODE[27997] := 16#8947;
   // GBK_TO_UNICODE[27998] := 16#D24E;
   // GBK_TO_UNICODE[27999] := 16#8948;
   // GBK_TO_UNICODE[28000] := 16#D24F;
   // GBK_TO_UNICODE[28001] := 16#8949;
   // GBK_TO_UNICODE[28002] := 16#D250;
   // GBK_TO_UNICODE[28003] := 16#894A;
   // GBK_TO_UNICODE[28004] := 16#D251;
   // GBK_TO_UNICODE[28005] := 16#894B;
   // GBK_TO_UNICODE[28006] := 16#D252;
   // GBK_TO_UNICODE[28007] := 16#894C;
   // GBK_TO_UNICODE[28008] := 16#D253;
   // GBK_TO_UNICODE[28009] := 16#894D;
   // GBK_TO_UNICODE[28010] := 16#D254;
   // GBK_TO_UNICODE[28011] := 16#894E;
   // GBK_TO_UNICODE[28012] := 16#D255;
   // GBK_TO_UNICODE[28013] := 16#894F;
   // GBK_TO_UNICODE[28014] := 16#D256;
   // GBK_TO_UNICODE[28015] := 16#8950;
   // GBK_TO_UNICODE[28016] := 16#D257;
   // GBK_TO_UNICODE[28017] := 16#8951;
   // GBK_TO_UNICODE[28018] := 16#D258;
   // GBK_TO_UNICODE[28019] := 16#8952;
   // GBK_TO_UNICODE[28020] := 16#D259;
   // GBK_TO_UNICODE[28021] := 16#8953;
   // GBK_TO_UNICODE[28022] := 16#D25A;
   // GBK_TO_UNICODE[28023] := 16#8954;
   // GBK_TO_UNICODE[28024] := 16#D25B;
   // GBK_TO_UNICODE[28025] := 16#8955;
   // GBK_TO_UNICODE[28026] := 16#D25C;
   // GBK_TO_UNICODE[28027] := 16#8956;
   // GBK_TO_UNICODE[28028] := 16#D25D;
   // GBK_TO_UNICODE[28029] := 16#8957;
   // GBK_TO_UNICODE[28030] := 16#D25E;
   // GBK_TO_UNICODE[28031] := 16#8958;
   // GBK_TO_UNICODE[28032] := 16#D25F;
   // GBK_TO_UNICODE[28033] := 16#8959;
   // GBK_TO_UNICODE[28034] := 16#D260;
   // GBK_TO_UNICODE[28035] := 16#895A;
   // GBK_TO_UNICODE[28036] := 16#D261;
   // GBK_TO_UNICODE[28037] := 16#895B;
   // GBK_TO_UNICODE[28038] := 16#D262;
   // GBK_TO_UNICODE[28039] := 16#895C;
   // GBK_TO_UNICODE[28040] := 16#D263;
   // GBK_TO_UNICODE[28041] := 16#895D;
   // GBK_TO_UNICODE[28042] := 16#D264;
   // GBK_TO_UNICODE[28043] := 16#8960;
   // GBK_TO_UNICODE[28044] := 16#D265;
   // GBK_TO_UNICODE[28045] := 16#8961;
   // GBK_TO_UNICODE[28046] := 16#D266;
   // GBK_TO_UNICODE[28047] := 16#8962;
   // GBK_TO_UNICODE[28048] := 16#D267;
   // GBK_TO_UNICODE[28049] := 16#8963;
   // GBK_TO_UNICODE[28050] := 16#D268;
   // GBK_TO_UNICODE[28051] := 16#8964;
   // GBK_TO_UNICODE[28052] := 16#D269;
   // GBK_TO_UNICODE[28053] := 16#8965;
   // GBK_TO_UNICODE[28054] := 16#D26A;
   // GBK_TO_UNICODE[28055] := 16#8967;
   // GBK_TO_UNICODE[28056] := 16#D26B;
   // GBK_TO_UNICODE[28057] := 16#8968;
   // GBK_TO_UNICODE[28058] := 16#D26C;
   // GBK_TO_UNICODE[28059] := 16#8969;
   // GBK_TO_UNICODE[28060] := 16#D26D;
   // GBK_TO_UNICODE[28061] := 16#896A;
   // GBK_TO_UNICODE[28062] := 16#D26E;
   // GBK_TO_UNICODE[28063] := 16#896B;
   // GBK_TO_UNICODE[28064] := 16#D26F;
   // GBK_TO_UNICODE[28065] := 16#896C;
   // GBK_TO_UNICODE[28066] := 16#D270;
   // GBK_TO_UNICODE[28067] := 16#896D;
   // GBK_TO_UNICODE[28068] := 16#D271;
   // GBK_TO_UNICODE[28069] := 16#896E;
   // GBK_TO_UNICODE[28070] := 16#D272;
   // GBK_TO_UNICODE[28071] := 16#896F;
   // GBK_TO_UNICODE[28072] := 16#D273;
   // GBK_TO_UNICODE[28073] := 16#8970;
   // GBK_TO_UNICODE[28074] := 16#D274;
   // GBK_TO_UNICODE[28075] := 16#8971;
   // GBK_TO_UNICODE[28076] := 16#D275;
   // GBK_TO_UNICODE[28077] := 16#8972;
   // GBK_TO_UNICODE[28078] := 16#D276;
   // GBK_TO_UNICODE[28079] := 16#8973;
   // GBK_TO_UNICODE[28080] := 16#D277;
   // GBK_TO_UNICODE[28081] := 16#8974;
   // GBK_TO_UNICODE[28082] := 16#D278;
   // GBK_TO_UNICODE[28083] := 16#8975;
   // GBK_TO_UNICODE[28084] := 16#D279;
   // GBK_TO_UNICODE[28085] := 16#8976;
   // GBK_TO_UNICODE[28086] := 16#D27A;
   // GBK_TO_UNICODE[28087] := 16#8977;
   // GBK_TO_UNICODE[28088] := 16#D27B;
   // GBK_TO_UNICODE[28089] := 16#8978;
   // GBK_TO_UNICODE[28090] := 16#D27C;
   // GBK_TO_UNICODE[28091] := 16#8979;
   // GBK_TO_UNICODE[28092] := 16#D27D;
   // GBK_TO_UNICODE[28093] := 16#897A;
   // GBK_TO_UNICODE[28094] := 16#D27E;
   // GBK_TO_UNICODE[28095] := 16#897C;
   // GBK_TO_UNICODE[28096] := 16#D280;
   // GBK_TO_UNICODE[28097] := 16#897D;
   // GBK_TO_UNICODE[28098] := 16#D281;
   // GBK_TO_UNICODE[28099] := 16#897E;
   // GBK_TO_UNICODE[28100] := 16#D282;
   // GBK_TO_UNICODE[28101] := 16#8980;
   // GBK_TO_UNICODE[28102] := 16#D283;
   // GBK_TO_UNICODE[28103] := 16#8982;
   // GBK_TO_UNICODE[28104] := 16#D284;
   // GBK_TO_UNICODE[28105] := 16#8984;
   // GBK_TO_UNICODE[28106] := 16#D285;
   // GBK_TO_UNICODE[28107] := 16#8985;
   // GBK_TO_UNICODE[28108] := 16#D286;
   // GBK_TO_UNICODE[28109] := 16#8987;
   // GBK_TO_UNICODE[28110] := 16#D287;
   // GBK_TO_UNICODE[28111] := 16#8988;
   // GBK_TO_UNICODE[28112] := 16#D288;
   // GBK_TO_UNICODE[28113] := 16#8989;
   // GBK_TO_UNICODE[28114] := 16#D289;
   // GBK_TO_UNICODE[28115] := 16#898A;
   // GBK_TO_UNICODE[28116] := 16#D28A;
   // GBK_TO_UNICODE[28117] := 16#898B;
   // GBK_TO_UNICODE[28118] := 16#D28B;
   // GBK_TO_UNICODE[28119] := 16#898C;
   // GBK_TO_UNICODE[28120] := 16#D28C;
   // GBK_TO_UNICODE[28121] := 16#898D;
   // GBK_TO_UNICODE[28122] := 16#D28D;
   // GBK_TO_UNICODE[28123] := 16#898E;
   // GBK_TO_UNICODE[28124] := 16#D28E;
   // GBK_TO_UNICODE[28125] := 16#898F;
   // GBK_TO_UNICODE[28126] := 16#D28F;
   // GBK_TO_UNICODE[28127] := 16#8990;
   // GBK_TO_UNICODE[28128] := 16#D290;
   // GBK_TO_UNICODE[28129] := 16#8991;
   // GBK_TO_UNICODE[28130] := 16#D291;
   // GBK_TO_UNICODE[28131] := 16#8992;
   // GBK_TO_UNICODE[28132] := 16#D292;
   // GBK_TO_UNICODE[28133] := 16#8993;
   // GBK_TO_UNICODE[28134] := 16#D293;
   // GBK_TO_UNICODE[28135] := 16#8994;
   // GBK_TO_UNICODE[28136] := 16#D294;
   // GBK_TO_UNICODE[28137] := 16#8995;
   // GBK_TO_UNICODE[28138] := 16#D295;
   // GBK_TO_UNICODE[28139] := 16#8996;
   // GBK_TO_UNICODE[28140] := 16#D296;
   // GBK_TO_UNICODE[28141] := 16#8997;
   // GBK_TO_UNICODE[28142] := 16#D297;
   // GBK_TO_UNICODE[28143] := 16#8998;
   // GBK_TO_UNICODE[28144] := 16#D298;
   // GBK_TO_UNICODE[28145] := 16#8999;
   // GBK_TO_UNICODE[28146] := 16#D299;
   // GBK_TO_UNICODE[28147] := 16#899A;
   // GBK_TO_UNICODE[28148] := 16#D29A;
   // GBK_TO_UNICODE[28149] := 16#899B;
   // GBK_TO_UNICODE[28150] := 16#D29B;
   // GBK_TO_UNICODE[28151] := 16#899C;
   // GBK_TO_UNICODE[28152] := 16#D29C;
   // GBK_TO_UNICODE[28153] := 16#899D;
   // GBK_TO_UNICODE[28154] := 16#D29D;
   // GBK_TO_UNICODE[28155] := 16#899E;
   // GBK_TO_UNICODE[28156] := 16#D29E;
   // GBK_TO_UNICODE[28157] := 16#899F;
   // GBK_TO_UNICODE[28158] := 16#D29F;
   // GBK_TO_UNICODE[28159] := 16#89A0;
   // GBK_TO_UNICODE[28160] := 16#D2A0;
   // GBK_TO_UNICODE[28161] := 16#89A1;
   // GBK_TO_UNICODE[28162] := 16#D2A1;
   // GBK_TO_UNICODE[28163] := 16#6447;
   // GBK_TO_UNICODE[28164] := 16#D2A2;
   // GBK_TO_UNICODE[28165] := 16#5C27;
   // GBK_TO_UNICODE[28166] := 16#D2A3;
   // GBK_TO_UNICODE[28167] := 16#9065;
   // GBK_TO_UNICODE[28168] := 16#D2A4;
   // GBK_TO_UNICODE[28169] := 16#7A91;
   // GBK_TO_UNICODE[28170] := 16#D2A5;
   // GBK_TO_UNICODE[28171] := 16#8C23;
   // GBK_TO_UNICODE[28172] := 16#D2A6;
   // GBK_TO_UNICODE[28173] := 16#59DA;
   // GBK_TO_UNICODE[28174] := 16#D2A7;
   // GBK_TO_UNICODE[28175] := 16#54AC;
   // GBK_TO_UNICODE[28176] := 16#D2A8;
   // GBK_TO_UNICODE[28177] := 16#8200;
   // GBK_TO_UNICODE[28178] := 16#D2A9;
   // GBK_TO_UNICODE[28179] := 16#836F;
   // GBK_TO_UNICODE[28180] := 16#D2AA;
   // GBK_TO_UNICODE[28181] := 16#8981;
   // GBK_TO_UNICODE[28182] := 16#D2AB;
   // GBK_TO_UNICODE[28183] := 16#8000;
   // GBK_TO_UNICODE[28184] := 16#D2AC;
   // GBK_TO_UNICODE[28185] := 16#6930;
   // GBK_TO_UNICODE[28186] := 16#D2AD;
   // GBK_TO_UNICODE[28187] := 16#564E;
   // GBK_TO_UNICODE[28188] := 16#D2AE;
   // GBK_TO_UNICODE[28189] := 16#8036;
   // GBK_TO_UNICODE[28190] := 16#D2AF;
   // GBK_TO_UNICODE[28191] := 16#7237;
   // GBK_TO_UNICODE[28192] := 16#D2B0;
   // GBK_TO_UNICODE[28193] := 16#91CE;
   // GBK_TO_UNICODE[28194] := 16#D2B1;
   // GBK_TO_UNICODE[28195] := 16#51B6;
   // GBK_TO_UNICODE[28196] := 16#D2B2;
   // GBK_TO_UNICODE[28197] := 16#4E5F;
   // GBK_TO_UNICODE[28198] := 16#D2B3;
   // GBK_TO_UNICODE[28199] := 16#9875;
   // GBK_TO_UNICODE[28200] := 16#D2B4;
   // GBK_TO_UNICODE[28201] := 16#6396;
   // GBK_TO_UNICODE[28202] := 16#D2B5;
   // GBK_TO_UNICODE[28203] := 16#4E1A;
   // GBK_TO_UNICODE[28204] := 16#D2B6;
   // GBK_TO_UNICODE[28205] := 16#53F6;
   // GBK_TO_UNICODE[28206] := 16#D2B7;
   // GBK_TO_UNICODE[28207] := 16#66F3;
   // GBK_TO_UNICODE[28208] := 16#D2B8;
   // GBK_TO_UNICODE[28209] := 16#814B;
   // GBK_TO_UNICODE[28210] := 16#D2B9;
   // GBK_TO_UNICODE[28211] := 16#591C;
   // GBK_TO_UNICODE[28212] := 16#D2BA;
   // GBK_TO_UNICODE[28213] := 16#6DB2;
   // GBK_TO_UNICODE[28214] := 16#D2BB;
   // GBK_TO_UNICODE[28215] := 16#4E00;
   // GBK_TO_UNICODE[28216] := 16#D2BC;
   // GBK_TO_UNICODE[28217] := 16#58F9;
   // GBK_TO_UNICODE[28218] := 16#D2BD;
   // GBK_TO_UNICODE[28219] := 16#533B;
   // GBK_TO_UNICODE[28220] := 16#D2BE;
   // GBK_TO_UNICODE[28221] := 16#63D6;
   // GBK_TO_UNICODE[28222] := 16#D2BF;
   // GBK_TO_UNICODE[28223] := 16#94F1;
   // GBK_TO_UNICODE[28224] := 16#D2C0;
   // GBK_TO_UNICODE[28225] := 16#4F9D;
   // GBK_TO_UNICODE[28226] := 16#D2C1;
   // GBK_TO_UNICODE[28227] := 16#4F0A;
   // GBK_TO_UNICODE[28228] := 16#D2C2;
   // GBK_TO_UNICODE[28229] := 16#8863;
   // GBK_TO_UNICODE[28230] := 16#D2C3;
   // GBK_TO_UNICODE[28231] := 16#9890;
   // GBK_TO_UNICODE[28232] := 16#D2C4;
   // GBK_TO_UNICODE[28233] := 16#5937;
   // GBK_TO_UNICODE[28234] := 16#D2C5;
   // GBK_TO_UNICODE[28235] := 16#9057;
   // GBK_TO_UNICODE[28236] := 16#D2C6;
   // GBK_TO_UNICODE[28237] := 16#79FB;
   // GBK_TO_UNICODE[28238] := 16#D2C7;
   // GBK_TO_UNICODE[28239] := 16#4EEA;
   // GBK_TO_UNICODE[28240] := 16#D2C8;
   // GBK_TO_UNICODE[28241] := 16#80F0;
   // GBK_TO_UNICODE[28242] := 16#D2C9;
   // GBK_TO_UNICODE[28243] := 16#7591;
   // GBK_TO_UNICODE[28244] := 16#D2CA;
   // GBK_TO_UNICODE[28245] := 16#6C82;
   // GBK_TO_UNICODE[28246] := 16#D2CB;
   // GBK_TO_UNICODE[28247] := 16#5B9C;
   // GBK_TO_UNICODE[28248] := 16#D2CC;
   // GBK_TO_UNICODE[28249] := 16#59E8;
   // GBK_TO_UNICODE[28250] := 16#D2CD;
   // GBK_TO_UNICODE[28251] := 16#5F5D;
   // GBK_TO_UNICODE[28252] := 16#D2CE;
   // GBK_TO_UNICODE[28253] := 16#6905;
   // GBK_TO_UNICODE[28254] := 16#D2CF;
   // GBK_TO_UNICODE[28255] := 16#8681;
   // GBK_TO_UNICODE[28256] := 16#D2D0;
   // GBK_TO_UNICODE[28257] := 16#501A;
   // GBK_TO_UNICODE[28258] := 16#D2D1;
   // GBK_TO_UNICODE[28259] := 16#5DF2;
   // GBK_TO_UNICODE[28260] := 16#D2D2;
   // GBK_TO_UNICODE[28261] := 16#4E59;
   // GBK_TO_UNICODE[28262] := 16#D2D3;
   // GBK_TO_UNICODE[28263] := 16#77E3;
   // GBK_TO_UNICODE[28264] := 16#D2D4;
   // GBK_TO_UNICODE[28265] := 16#4EE5;
   // GBK_TO_UNICODE[28266] := 16#D2D5;
   // GBK_TO_UNICODE[28267] := 16#827A;
   // GBK_TO_UNICODE[28268] := 16#D2D6;
   // GBK_TO_UNICODE[28269] := 16#6291;
   // GBK_TO_UNICODE[28270] := 16#D2D7;
   // GBK_TO_UNICODE[28271] := 16#6613;
   // GBK_TO_UNICODE[28272] := 16#D2D8;
   // GBK_TO_UNICODE[28273] := 16#9091;
   // GBK_TO_UNICODE[28274] := 16#D2D9;
   // GBK_TO_UNICODE[28275] := 16#5C79;
   // GBK_TO_UNICODE[28276] := 16#D2DA;
   // GBK_TO_UNICODE[28277] := 16#4EBF;
   // GBK_TO_UNICODE[28278] := 16#D2DB;
   // GBK_TO_UNICODE[28279] := 16#5F79;
   // GBK_TO_UNICODE[28280] := 16#D2DC;
   // GBK_TO_UNICODE[28281] := 16#81C6;
   // GBK_TO_UNICODE[28282] := 16#D2DD;
   // GBK_TO_UNICODE[28283] := 16#9038;
   // GBK_TO_UNICODE[28284] := 16#D2DE;
   // GBK_TO_UNICODE[28285] := 16#8084;
   // GBK_TO_UNICODE[28286] := 16#D2DF;
   // GBK_TO_UNICODE[28287] := 16#75AB;
   // GBK_TO_UNICODE[28288] := 16#D2E0;
   // GBK_TO_UNICODE[28289] := 16#4EA6;
   // GBK_TO_UNICODE[28290] := 16#D2E1;
   // GBK_TO_UNICODE[28291] := 16#88D4;
   // GBK_TO_UNICODE[28292] := 16#D2E2;
   // GBK_TO_UNICODE[28293] := 16#610F;
   // GBK_TO_UNICODE[28294] := 16#D2E3;
   // GBK_TO_UNICODE[28295] := 16#6BC5;
   // GBK_TO_UNICODE[28296] := 16#D2E4;
   // GBK_TO_UNICODE[28297] := 16#5FC6;
   // GBK_TO_UNICODE[28298] := 16#D2E5;
   // GBK_TO_UNICODE[28299] := 16#4E49;
   // GBK_TO_UNICODE[28300] := 16#D2E6;
   // GBK_TO_UNICODE[28301] := 16#76CA;
   // GBK_TO_UNICODE[28302] := 16#D2E7;
   // GBK_TO_UNICODE[28303] := 16#6EA2;
   // GBK_TO_UNICODE[28304] := 16#D2E8;
   // GBK_TO_UNICODE[28305] := 16#8BE3;
   // GBK_TO_UNICODE[28306] := 16#D2E9;
   // GBK_TO_UNICODE[28307] := 16#8BAE;
   // GBK_TO_UNICODE[28308] := 16#D2EA;
   // GBK_TO_UNICODE[28309] := 16#8C0A;
   // GBK_TO_UNICODE[28310] := 16#D2EB;
   // GBK_TO_UNICODE[28311] := 16#8BD1;
   // GBK_TO_UNICODE[28312] := 16#D2EC;
   // GBK_TO_UNICODE[28313] := 16#5F02;
   // GBK_TO_UNICODE[28314] := 16#D2ED;
   // GBK_TO_UNICODE[28315] := 16#7FFC;
   // GBK_TO_UNICODE[28316] := 16#D2EE;
   // GBK_TO_UNICODE[28317] := 16#7FCC;
   // GBK_TO_UNICODE[28318] := 16#D2EF;
   // GBK_TO_UNICODE[28319] := 16#7ECE;
   // GBK_TO_UNICODE[28320] := 16#D2F0;
   // GBK_TO_UNICODE[28321] := 16#8335;
   // GBK_TO_UNICODE[28322] := 16#D2F1;
   // GBK_TO_UNICODE[28323] := 16#836B;
   // GBK_TO_UNICODE[28324] := 16#D2F2;
   // GBK_TO_UNICODE[28325] := 16#56E0;
   // GBK_TO_UNICODE[28326] := 16#D2F3;
   // GBK_TO_UNICODE[28327] := 16#6BB7;
   // GBK_TO_UNICODE[28328] := 16#D2F4;
   // GBK_TO_UNICODE[28329] := 16#97F3;
   // GBK_TO_UNICODE[28330] := 16#D2F5;
   // GBK_TO_UNICODE[28331] := 16#9634;
   // GBK_TO_UNICODE[28332] := 16#D2F6;
   // GBK_TO_UNICODE[28333] := 16#59FB;
   // GBK_TO_UNICODE[28334] := 16#D2F7;
   // GBK_TO_UNICODE[28335] := 16#541F;
   // GBK_TO_UNICODE[28336] := 16#D2F8;
   // GBK_TO_UNICODE[28337] := 16#94F6;
   // GBK_TO_UNICODE[28338] := 16#D2F9;
   // GBK_TO_UNICODE[28339] := 16#6DEB;
   // GBK_TO_UNICODE[28340] := 16#D2FA;
   // GBK_TO_UNICODE[28341] := 16#5BC5;
   // GBK_TO_UNICODE[28342] := 16#D2FB;
   // GBK_TO_UNICODE[28343] := 16#996E;
   // GBK_TO_UNICODE[28344] := 16#D2FC;
   // GBK_TO_UNICODE[28345] := 16#5C39;
   // GBK_TO_UNICODE[28346] := 16#D2FD;
   // GBK_TO_UNICODE[28347] := 16#5F15;
   // GBK_TO_UNICODE[28348] := 16#D2FE;
   // GBK_TO_UNICODE[28349] := 16#9690;
   // GBK_TO_UNICODE[28350] := 16#D340;
   // GBK_TO_UNICODE[28351] := 16#89A2;
   // GBK_TO_UNICODE[28352] := 16#D341;
   // GBK_TO_UNICODE[28353] := 16#89A3;
   // GBK_TO_UNICODE[28354] := 16#D342;
   // GBK_TO_UNICODE[28355] := 16#89A4;
   // GBK_TO_UNICODE[28356] := 16#D343;
   // GBK_TO_UNICODE[28357] := 16#89A5;
   // GBK_TO_UNICODE[28358] := 16#D344;
   // GBK_TO_UNICODE[28359] := 16#89A6;
   // GBK_TO_UNICODE[28360] := 16#D345;
   // GBK_TO_UNICODE[28361] := 16#89A7;
   // GBK_TO_UNICODE[28362] := 16#D346;
   // GBK_TO_UNICODE[28363] := 16#89A8;
   // GBK_TO_UNICODE[28364] := 16#D347;
   // GBK_TO_UNICODE[28365] := 16#89A9;
   // GBK_TO_UNICODE[28366] := 16#D348;
   // GBK_TO_UNICODE[28367] := 16#89AA;
   // GBK_TO_UNICODE[28368] := 16#D349;
   // GBK_TO_UNICODE[28369] := 16#89AB;
   // GBK_TO_UNICODE[28370] := 16#D34A;
   // GBK_TO_UNICODE[28371] := 16#89AC;
   // GBK_TO_UNICODE[28372] := 16#D34B;
   // GBK_TO_UNICODE[28373] := 16#89AD;
   // GBK_TO_UNICODE[28374] := 16#D34C;
   // GBK_TO_UNICODE[28375] := 16#89AE;
   // GBK_TO_UNICODE[28376] := 16#D34D;
   // GBK_TO_UNICODE[28377] := 16#89AF;
   // GBK_TO_UNICODE[28378] := 16#D34E;
   // GBK_TO_UNICODE[28379] := 16#89B0;
   // GBK_TO_UNICODE[28380] := 16#D34F;
   // GBK_TO_UNICODE[28381] := 16#89B1;
   // GBK_TO_UNICODE[28382] := 16#D350;
   // GBK_TO_UNICODE[28383] := 16#89B2;
   // GBK_TO_UNICODE[28384] := 16#D351;
   // GBK_TO_UNICODE[28385] := 16#89B3;
   // GBK_TO_UNICODE[28386] := 16#D352;
   // GBK_TO_UNICODE[28387] := 16#89B4;
   // GBK_TO_UNICODE[28388] := 16#D353;
   // GBK_TO_UNICODE[28389] := 16#89B5;
   // GBK_TO_UNICODE[28390] := 16#D354;
   // GBK_TO_UNICODE[28391] := 16#89B6;
   // GBK_TO_UNICODE[28392] := 16#D355;
   // GBK_TO_UNICODE[28393] := 16#89B7;
   // GBK_TO_UNICODE[28394] := 16#D356;
   // GBK_TO_UNICODE[28395] := 16#89B8;
   // GBK_TO_UNICODE[28396] := 16#D357;
   // GBK_TO_UNICODE[28397] := 16#89B9;
   // GBK_TO_UNICODE[28398] := 16#D358;
   // GBK_TO_UNICODE[28399] := 16#89BA;
   // GBK_TO_UNICODE[28400] := 16#D359;
   // GBK_TO_UNICODE[28401] := 16#89BB;
   // GBK_TO_UNICODE[28402] := 16#D35A;
   // GBK_TO_UNICODE[28403] := 16#89BC;
   // GBK_TO_UNICODE[28404] := 16#D35B;
   // GBK_TO_UNICODE[28405] := 16#89BD;
   // GBK_TO_UNICODE[28406] := 16#D35C;
   // GBK_TO_UNICODE[28407] := 16#89BE;
   // GBK_TO_UNICODE[28408] := 16#D35D;
   // GBK_TO_UNICODE[28409] := 16#89BF;
   // GBK_TO_UNICODE[28410] := 16#D35E;
   // GBK_TO_UNICODE[28411] := 16#89C0;
   // GBK_TO_UNICODE[28412] := 16#D35F;
   // GBK_TO_UNICODE[28413] := 16#89C3;
   // GBK_TO_UNICODE[28414] := 16#D360;
   // GBK_TO_UNICODE[28415] := 16#89CD;
   // GBK_TO_UNICODE[28416] := 16#D361;
   // GBK_TO_UNICODE[28417] := 16#89D3;
   // GBK_TO_UNICODE[28418] := 16#D362;
   // GBK_TO_UNICODE[28419] := 16#89D4;
   // GBK_TO_UNICODE[28420] := 16#D363;
   // GBK_TO_UNICODE[28421] := 16#89D5;
   // GBK_TO_UNICODE[28422] := 16#D364;
   // GBK_TO_UNICODE[28423] := 16#89D7;
   // GBK_TO_UNICODE[28424] := 16#D365;
   // GBK_TO_UNICODE[28425] := 16#89D8;
   // GBK_TO_UNICODE[28426] := 16#D366;
   // GBK_TO_UNICODE[28427] := 16#89D9;
   // GBK_TO_UNICODE[28428] := 16#D367;
   // GBK_TO_UNICODE[28429] := 16#89DB;
   // GBK_TO_UNICODE[28430] := 16#D368;
   // GBK_TO_UNICODE[28431] := 16#89DD;
   // GBK_TO_UNICODE[28432] := 16#D369;
   // GBK_TO_UNICODE[28433] := 16#89DF;
   // GBK_TO_UNICODE[28434] := 16#D36A;
   // GBK_TO_UNICODE[28435] := 16#89E0;
   // GBK_TO_UNICODE[28436] := 16#D36B;
   // GBK_TO_UNICODE[28437] := 16#89E1;
   // GBK_TO_UNICODE[28438] := 16#D36C;
   // GBK_TO_UNICODE[28439] := 16#89E2;
   // GBK_TO_UNICODE[28440] := 16#D36D;
   // GBK_TO_UNICODE[28441] := 16#89E4;
   // GBK_TO_UNICODE[28442] := 16#D36E;
   // GBK_TO_UNICODE[28443] := 16#89E7;
   // GBK_TO_UNICODE[28444] := 16#D36F;
   // GBK_TO_UNICODE[28445] := 16#89E8;
   // GBK_TO_UNICODE[28446] := 16#D370;
   // GBK_TO_UNICODE[28447] := 16#89E9;
   // GBK_TO_UNICODE[28448] := 16#D371;
   // GBK_TO_UNICODE[28449] := 16#89EA;
   // GBK_TO_UNICODE[28450] := 16#D372;
   // GBK_TO_UNICODE[28451] := 16#89EC;
   // GBK_TO_UNICODE[28452] := 16#D373;
   // GBK_TO_UNICODE[28453] := 16#89ED;
   // GBK_TO_UNICODE[28454] := 16#D374;
   // GBK_TO_UNICODE[28455] := 16#89EE;
   // GBK_TO_UNICODE[28456] := 16#D375;
   // GBK_TO_UNICODE[28457] := 16#89F0;
   // GBK_TO_UNICODE[28458] := 16#D376;
   // GBK_TO_UNICODE[28459] := 16#89F1;
   // GBK_TO_UNICODE[28460] := 16#D377;
   // GBK_TO_UNICODE[28461] := 16#89F2;
   // GBK_TO_UNICODE[28462] := 16#D378;
   // GBK_TO_UNICODE[28463] := 16#89F4;
   // GBK_TO_UNICODE[28464] := 16#D379;
   // GBK_TO_UNICODE[28465] := 16#89F5;
   // GBK_TO_UNICODE[28466] := 16#D37A;
   // GBK_TO_UNICODE[28467] := 16#89F6;
   // GBK_TO_UNICODE[28468] := 16#D37B;
   // GBK_TO_UNICODE[28469] := 16#89F7;
   // GBK_TO_UNICODE[28470] := 16#D37C;
   // GBK_TO_UNICODE[28471] := 16#89F8;
   // GBK_TO_UNICODE[28472] := 16#D37D;
   // GBK_TO_UNICODE[28473] := 16#89F9;
   // GBK_TO_UNICODE[28474] := 16#D37E;
   // GBK_TO_UNICODE[28475] := 16#89FA;
   // GBK_TO_UNICODE[28476] := 16#D380;
   // GBK_TO_UNICODE[28477] := 16#89FB;
   // GBK_TO_UNICODE[28478] := 16#D381;
   // GBK_TO_UNICODE[28479] := 16#89FC;
   // GBK_TO_UNICODE[28480] := 16#D382;
   // GBK_TO_UNICODE[28481] := 16#89FD;
   // GBK_TO_UNICODE[28482] := 16#D383;
   // GBK_TO_UNICODE[28483] := 16#89FE;
   // GBK_TO_UNICODE[28484] := 16#D384;
   // GBK_TO_UNICODE[28485] := 16#89FF;
   // GBK_TO_UNICODE[28486] := 16#D385;
   // GBK_TO_UNICODE[28487] := 16#8A01;
   // GBK_TO_UNICODE[28488] := 16#D386;
   // GBK_TO_UNICODE[28489] := 16#8A02;
   // GBK_TO_UNICODE[28490] := 16#D387;
   // GBK_TO_UNICODE[28491] := 16#8A03;
   // GBK_TO_UNICODE[28492] := 16#D388;
   // GBK_TO_UNICODE[28493] := 16#8A04;
   // GBK_TO_UNICODE[28494] := 16#D389;
   // GBK_TO_UNICODE[28495] := 16#8A05;
   // GBK_TO_UNICODE[28496] := 16#D38A;
   // GBK_TO_UNICODE[28497] := 16#8A06;
   // GBK_TO_UNICODE[28498] := 16#D38B;
   // GBK_TO_UNICODE[28499] := 16#8A08;
   // GBK_TO_UNICODE[28500] := 16#D38C;
   // GBK_TO_UNICODE[28501] := 16#8A09;
   // GBK_TO_UNICODE[28502] := 16#D38D;
   // GBK_TO_UNICODE[28503] := 16#8A0A;
   // GBK_TO_UNICODE[28504] := 16#D38E;
   // GBK_TO_UNICODE[28505] := 16#8A0B;
   // GBK_TO_UNICODE[28506] := 16#D38F;
   // GBK_TO_UNICODE[28507] := 16#8A0C;
   // GBK_TO_UNICODE[28508] := 16#D390;
   // GBK_TO_UNICODE[28509] := 16#8A0D;
   // GBK_TO_UNICODE[28510] := 16#D391;
   // GBK_TO_UNICODE[28511] := 16#8A0E;
   // GBK_TO_UNICODE[28512] := 16#D392;
   // GBK_TO_UNICODE[28513] := 16#8A0F;
   // GBK_TO_UNICODE[28514] := 16#D393;
   // GBK_TO_UNICODE[28515] := 16#8A10;
   // GBK_TO_UNICODE[28516] := 16#D394;
   // GBK_TO_UNICODE[28517] := 16#8A11;
   // GBK_TO_UNICODE[28518] := 16#D395;
   // GBK_TO_UNICODE[28519] := 16#8A12;
   // GBK_TO_UNICODE[28520] := 16#D396;
   // GBK_TO_UNICODE[28521] := 16#8A13;
   // GBK_TO_UNICODE[28522] := 16#D397;
   // GBK_TO_UNICODE[28523] := 16#8A14;
   // GBK_TO_UNICODE[28524] := 16#D398;
   // GBK_TO_UNICODE[28525] := 16#8A15;
   // GBK_TO_UNICODE[28526] := 16#D399;
   // GBK_TO_UNICODE[28527] := 16#8A16;
   // GBK_TO_UNICODE[28528] := 16#D39A;
   // GBK_TO_UNICODE[28529] := 16#8A17;
   // GBK_TO_UNICODE[28530] := 16#D39B;
   // GBK_TO_UNICODE[28531] := 16#8A18;
   // GBK_TO_UNICODE[28532] := 16#D39C;
   // GBK_TO_UNICODE[28533] := 16#8A19;
   // GBK_TO_UNICODE[28534] := 16#D39D;
   // GBK_TO_UNICODE[28535] := 16#8A1A;
   // GBK_TO_UNICODE[28536] := 16#D39E;
   // GBK_TO_UNICODE[28537] := 16#8A1B;
   // GBK_TO_UNICODE[28538] := 16#D39F;
   // GBK_TO_UNICODE[28539] := 16#8A1C;
   // GBK_TO_UNICODE[28540] := 16#D3A0;
   // GBK_TO_UNICODE[28541] := 16#8A1D;
   // GBK_TO_UNICODE[28542] := 16#D3A1;
   // GBK_TO_UNICODE[28543] := 16#5370;
   // GBK_TO_UNICODE[28544] := 16#D3A2;
   // GBK_TO_UNICODE[28545] := 16#82F1;
   // GBK_TO_UNICODE[28546] := 16#D3A3;
   // GBK_TO_UNICODE[28547] := 16#6A31;
   // GBK_TO_UNICODE[28548] := 16#D3A4;
   // GBK_TO_UNICODE[28549] := 16#5A74;
   // GBK_TO_UNICODE[28550] := 16#D3A5;
   // GBK_TO_UNICODE[28551] := 16#9E70;
   // GBK_TO_UNICODE[28552] := 16#D3A6;
   // GBK_TO_UNICODE[28553] := 16#5E94;
   // GBK_TO_UNICODE[28554] := 16#D3A7;
   // GBK_TO_UNICODE[28555] := 16#7F28;
   // GBK_TO_UNICODE[28556] := 16#D3A8;
   // GBK_TO_UNICODE[28557] := 16#83B9;
   // GBK_TO_UNICODE[28558] := 16#D3A9;
   // GBK_TO_UNICODE[28559] := 16#8424;
   // GBK_TO_UNICODE[28560] := 16#D3AA;
   // GBK_TO_UNICODE[28561] := 16#8425;
   // GBK_TO_UNICODE[28562] := 16#D3AB;
   // GBK_TO_UNICODE[28563] := 16#8367;
   // GBK_TO_UNICODE[28564] := 16#D3AC;
   // GBK_TO_UNICODE[28565] := 16#8747;
   // GBK_TO_UNICODE[28566] := 16#D3AD;
   // GBK_TO_UNICODE[28567] := 16#8FCE;
   // GBK_TO_UNICODE[28568] := 16#D3AE;
   // GBK_TO_UNICODE[28569] := 16#8D62;
   // GBK_TO_UNICODE[28570] := 16#D3AF;
   // GBK_TO_UNICODE[28571] := 16#76C8;
   // GBK_TO_UNICODE[28572] := 16#D3B0;
   // GBK_TO_UNICODE[28573] := 16#5F71;
   // GBK_TO_UNICODE[28574] := 16#D3B1;
   // GBK_TO_UNICODE[28575] := 16#9896;
   // GBK_TO_UNICODE[28576] := 16#D3B2;
   // GBK_TO_UNICODE[28577] := 16#786C;
   // GBK_TO_UNICODE[28578] := 16#D3B3;
   // GBK_TO_UNICODE[28579] := 16#6620;
   // GBK_TO_UNICODE[28580] := 16#D3B4;
   // GBK_TO_UNICODE[28581] := 16#54DF;
   // GBK_TO_UNICODE[28582] := 16#D3B5;
   // GBK_TO_UNICODE[28583] := 16#62E5;
   // GBK_TO_UNICODE[28584] := 16#D3B6;
   // GBK_TO_UNICODE[28585] := 16#4F63;
   // GBK_TO_UNICODE[28586] := 16#D3B7;
   // GBK_TO_UNICODE[28587] := 16#81C3;
   // GBK_TO_UNICODE[28588] := 16#D3B8;
   // GBK_TO_UNICODE[28589] := 16#75C8;
   // GBK_TO_UNICODE[28590] := 16#D3B9;
   // GBK_TO_UNICODE[28591] := 16#5EB8;
   // GBK_TO_UNICODE[28592] := 16#D3BA;
   // GBK_TO_UNICODE[28593] := 16#96CD;
   // GBK_TO_UNICODE[28594] := 16#D3BB;
   // GBK_TO_UNICODE[28595] := 16#8E0A;
   // GBK_TO_UNICODE[28596] := 16#D3BC;
   // GBK_TO_UNICODE[28597] := 16#86F9;
   // GBK_TO_UNICODE[28598] := 16#D3BD;
   // GBK_TO_UNICODE[28599] := 16#548F;
   // GBK_TO_UNICODE[28600] := 16#D3BE;
   // GBK_TO_UNICODE[28601] := 16#6CF3;
   // GBK_TO_UNICODE[28602] := 16#D3BF;
   // GBK_TO_UNICODE[28603] := 16#6D8C;
   // GBK_TO_UNICODE[28604] := 16#D3C0;
   // GBK_TO_UNICODE[28605] := 16#6C38;
   // GBK_TO_UNICODE[28606] := 16#D3C1;
   // GBK_TO_UNICODE[28607] := 16#607F;
   // GBK_TO_UNICODE[28608] := 16#D3C2;
   // GBK_TO_UNICODE[28609] := 16#52C7;
   // GBK_TO_UNICODE[28610] := 16#D3C3;
   // GBK_TO_UNICODE[28611] := 16#7528;
   // GBK_TO_UNICODE[28612] := 16#D3C4;
   // GBK_TO_UNICODE[28613] := 16#5E7D;
   // GBK_TO_UNICODE[28614] := 16#D3C5;
   // GBK_TO_UNICODE[28615] := 16#4F18;
   // GBK_TO_UNICODE[28616] := 16#D3C6;
   // GBK_TO_UNICODE[28617] := 16#60A0;
   // GBK_TO_UNICODE[28618] := 16#D3C7;
   // GBK_TO_UNICODE[28619] := 16#5FE7;
   // GBK_TO_UNICODE[28620] := 16#D3C8;
   // GBK_TO_UNICODE[28621] := 16#5C24;
   // GBK_TO_UNICODE[28622] := 16#D3C9;
   // GBK_TO_UNICODE[28623] := 16#7531;
   // GBK_TO_UNICODE[28624] := 16#D3CA;
   // GBK_TO_UNICODE[28625] := 16#90AE;
   // GBK_TO_UNICODE[28626] := 16#D3CB;
   // GBK_TO_UNICODE[28627] := 16#94C0;
   // GBK_TO_UNICODE[28628] := 16#D3CC;
   // GBK_TO_UNICODE[28629] := 16#72B9;
   // GBK_TO_UNICODE[28630] := 16#D3CD;
   // GBK_TO_UNICODE[28631] := 16#6CB9;
   // GBK_TO_UNICODE[28632] := 16#D3CE;
   // GBK_TO_UNICODE[28633] := 16#6E38;
   // GBK_TO_UNICODE[28634] := 16#D3CF;
   // GBK_TO_UNICODE[28635] := 16#9149;
   // GBK_TO_UNICODE[28636] := 16#D3D0;
   // GBK_TO_UNICODE[28637] := 16#6709;
   // GBK_TO_UNICODE[28638] := 16#D3D1;
   // GBK_TO_UNICODE[28639] := 16#53CB;
   // GBK_TO_UNICODE[28640] := 16#D3D2;
   // GBK_TO_UNICODE[28641] := 16#53F3;
   // GBK_TO_UNICODE[28642] := 16#D3D3;
   // GBK_TO_UNICODE[28643] := 16#4F51;
   // GBK_TO_UNICODE[28644] := 16#D3D4;
   // GBK_TO_UNICODE[28645] := 16#91C9;
   // GBK_TO_UNICODE[28646] := 16#D3D5;
   // GBK_TO_UNICODE[28647] := 16#8BF1;
   // GBK_TO_UNICODE[28648] := 16#D3D6;
   // GBK_TO_UNICODE[28649] := 16#53C8;
   // GBK_TO_UNICODE[28650] := 16#D3D7;
   // GBK_TO_UNICODE[28651] := 16#5E7C;
   // GBK_TO_UNICODE[28652] := 16#D3D8;
   // GBK_TO_UNICODE[28653] := 16#8FC2;
   // GBK_TO_UNICODE[28654] := 16#D3D9;
   // GBK_TO_UNICODE[28655] := 16#6DE4;
   // GBK_TO_UNICODE[28656] := 16#D3DA;
   // GBK_TO_UNICODE[28657] := 16#4E8E;
   // GBK_TO_UNICODE[28658] := 16#D3DB;
   // GBK_TO_UNICODE[28659] := 16#76C2;
   // GBK_TO_UNICODE[28660] := 16#D3DC;
   // GBK_TO_UNICODE[28661] := 16#6986;
   // GBK_TO_UNICODE[28662] := 16#D3DD;
   // GBK_TO_UNICODE[28663] := 16#865E;
   // GBK_TO_UNICODE[28664] := 16#D3DE;
   // GBK_TO_UNICODE[28665] := 16#611A;
   // GBK_TO_UNICODE[28666] := 16#D3DF;
   // GBK_TO_UNICODE[28667] := 16#8206;
   // GBK_TO_UNICODE[28668] := 16#D3E0;
   // GBK_TO_UNICODE[28669] := 16#4F59;
   // GBK_TO_UNICODE[28670] := 16#D3E1;
   // GBK_TO_UNICODE[28671] := 16#4FDE;
   // GBK_TO_UNICODE[28672] := 16#D3E2;
   // GBK_TO_UNICODE[28673] := 16#903E;
   // GBK_TO_UNICODE[28674] := 16#D3E3;
   // GBK_TO_UNICODE[28675] := 16#9C7C;
   // GBK_TO_UNICODE[28676] := 16#D3E4;
   // GBK_TO_UNICODE[28677] := 16#6109;
   // GBK_TO_UNICODE[28678] := 16#D3E5;
   // GBK_TO_UNICODE[28679] := 16#6E1D;
   // GBK_TO_UNICODE[28680] := 16#D3E6;
   // GBK_TO_UNICODE[28681] := 16#6E14;
   // GBK_TO_UNICODE[28682] := 16#D3E7;
   // GBK_TO_UNICODE[28683] := 16#9685;
   // GBK_TO_UNICODE[28684] := 16#D3E8;
   // GBK_TO_UNICODE[28685] := 16#4E88;
   // GBK_TO_UNICODE[28686] := 16#D3E9;
   // GBK_TO_UNICODE[28687] := 16#5A31;
   // GBK_TO_UNICODE[28688] := 16#D3EA;
   // GBK_TO_UNICODE[28689] := 16#96E8;
   // GBK_TO_UNICODE[28690] := 16#D3EB;
   // GBK_TO_UNICODE[28691] := 16#4E0E;
   // GBK_TO_UNICODE[28692] := 16#D3EC;
   // GBK_TO_UNICODE[28693] := 16#5C7F;
   // GBK_TO_UNICODE[28694] := 16#D3ED;
   // GBK_TO_UNICODE[28695] := 16#79B9;
   // GBK_TO_UNICODE[28696] := 16#D3EE;
   // GBK_TO_UNICODE[28697] := 16#5B87;
   // GBK_TO_UNICODE[28698] := 16#D3EF;
   // GBK_TO_UNICODE[28699] := 16#8BED;
   // GBK_TO_UNICODE[28700] := 16#D3F0;
   // GBK_TO_UNICODE[28701] := 16#7FBD;
   // GBK_TO_UNICODE[28702] := 16#D3F1;
   // GBK_TO_UNICODE[28703] := 16#7389;
   // GBK_TO_UNICODE[28704] := 16#D3F2;
   // GBK_TO_UNICODE[28705] := 16#57DF;
   // GBK_TO_UNICODE[28706] := 16#D3F3;
   // GBK_TO_UNICODE[28707] := 16#828B;
   // GBK_TO_UNICODE[28708] := 16#D3F4;
   // GBK_TO_UNICODE[28709] := 16#90C1;
   // GBK_TO_UNICODE[28710] := 16#D3F5;
   // GBK_TO_UNICODE[28711] := 16#5401;
   // GBK_TO_UNICODE[28712] := 16#D3F6;
   // GBK_TO_UNICODE[28713] := 16#9047;
   // GBK_TO_UNICODE[28714] := 16#D3F7;
   // GBK_TO_UNICODE[28715] := 16#55BB;
   // GBK_TO_UNICODE[28716] := 16#D3F8;
   // GBK_TO_UNICODE[28717] := 16#5CEA;
   // GBK_TO_UNICODE[28718] := 16#D3F9;
   // GBK_TO_UNICODE[28719] := 16#5FA1;
   // GBK_TO_UNICODE[28720] := 16#D3FA;
   // GBK_TO_UNICODE[28721] := 16#6108;
   // GBK_TO_UNICODE[28722] := 16#D3FB;
   // GBK_TO_UNICODE[28723] := 16#6B32;
   // GBK_TO_UNICODE[28724] := 16#D3FC;
   // GBK_TO_UNICODE[28725] := 16#72F1;
   // GBK_TO_UNICODE[28726] := 16#D3FD;
   // GBK_TO_UNICODE[28727] := 16#80B2;
   // GBK_TO_UNICODE[28728] := 16#D3FE;
   // GBK_TO_UNICODE[28729] := 16#8A89;
   // GBK_TO_UNICODE[28730] := 16#D440;
   // GBK_TO_UNICODE[28731] := 16#8A1E;
   // GBK_TO_UNICODE[28732] := 16#D441;
   // GBK_TO_UNICODE[28733] := 16#8A1F;
   // GBK_TO_UNICODE[28734] := 16#D442;
   // GBK_TO_UNICODE[28735] := 16#8A20;
   // GBK_TO_UNICODE[28736] := 16#D443;
   // GBK_TO_UNICODE[28737] := 16#8A21;
   // GBK_TO_UNICODE[28738] := 16#D444;
   // GBK_TO_UNICODE[28739] := 16#8A22;
   // GBK_TO_UNICODE[28740] := 16#D445;
   // GBK_TO_UNICODE[28741] := 16#8A23;
   // GBK_TO_UNICODE[28742] := 16#D446;
   // GBK_TO_UNICODE[28743] := 16#8A24;
   // GBK_TO_UNICODE[28744] := 16#D447;
   // GBK_TO_UNICODE[28745] := 16#8A25;
   // GBK_TO_UNICODE[28746] := 16#D448;
   // GBK_TO_UNICODE[28747] := 16#8A26;
   // GBK_TO_UNICODE[28748] := 16#D449;
   // GBK_TO_UNICODE[28749] := 16#8A27;
   // GBK_TO_UNICODE[28750] := 16#D44A;
   // GBK_TO_UNICODE[28751] := 16#8A28;
   // GBK_TO_UNICODE[28752] := 16#D44B;
   // GBK_TO_UNICODE[28753] := 16#8A29;
   // GBK_TO_UNICODE[28754] := 16#D44C;
   // GBK_TO_UNICODE[28755] := 16#8A2A;
   // GBK_TO_UNICODE[28756] := 16#D44D;
   // GBK_TO_UNICODE[28757] := 16#8A2B;
   // GBK_TO_UNICODE[28758] := 16#D44E;
   // GBK_TO_UNICODE[28759] := 16#8A2C;
   // GBK_TO_UNICODE[28760] := 16#D44F;
   // GBK_TO_UNICODE[28761] := 16#8A2D;
   // GBK_TO_UNICODE[28762] := 16#D450;
   // GBK_TO_UNICODE[28763] := 16#8A2E;
   // GBK_TO_UNICODE[28764] := 16#D451;
   // GBK_TO_UNICODE[28765] := 16#8A2F;
   // GBK_TO_UNICODE[28766] := 16#D452;
   // GBK_TO_UNICODE[28767] := 16#8A30;
   // GBK_TO_UNICODE[28768] := 16#D453;
   // GBK_TO_UNICODE[28769] := 16#8A31;
   // GBK_TO_UNICODE[28770] := 16#D454;
   // GBK_TO_UNICODE[28771] := 16#8A32;
   // GBK_TO_UNICODE[28772] := 16#D455;
   // GBK_TO_UNICODE[28773] := 16#8A33;
   // GBK_TO_UNICODE[28774] := 16#D456;
   // GBK_TO_UNICODE[28775] := 16#8A34;
   // GBK_TO_UNICODE[28776] := 16#D457;
   // GBK_TO_UNICODE[28777] := 16#8A35;
   // GBK_TO_UNICODE[28778] := 16#D458;
   // GBK_TO_UNICODE[28779] := 16#8A36;
   // GBK_TO_UNICODE[28780] := 16#D459;
   // GBK_TO_UNICODE[28781] := 16#8A37;
   // GBK_TO_UNICODE[28782] := 16#D45A;
   // GBK_TO_UNICODE[28783] := 16#8A38;
   // GBK_TO_UNICODE[28784] := 16#D45B;
   // GBK_TO_UNICODE[28785] := 16#8A39;
   // GBK_TO_UNICODE[28786] := 16#D45C;
   // GBK_TO_UNICODE[28787] := 16#8A3A;
   // GBK_TO_UNICODE[28788] := 16#D45D;
   // GBK_TO_UNICODE[28789] := 16#8A3B;
   // GBK_TO_UNICODE[28790] := 16#D45E;
   // GBK_TO_UNICODE[28791] := 16#8A3C;
   // GBK_TO_UNICODE[28792] := 16#D45F;
   // GBK_TO_UNICODE[28793] := 16#8A3D;
   // GBK_TO_UNICODE[28794] := 16#D460;
   // GBK_TO_UNICODE[28795] := 16#8A3F;
   // GBK_TO_UNICODE[28796] := 16#D461;
   // GBK_TO_UNICODE[28797] := 16#8A40;
   // GBK_TO_UNICODE[28798] := 16#D462;
   // GBK_TO_UNICODE[28799] := 16#8A41;
   // GBK_TO_UNICODE[28800] := 16#D463;
   // GBK_TO_UNICODE[28801] := 16#8A42;
   // GBK_TO_UNICODE[28802] := 16#D464;
   // GBK_TO_UNICODE[28803] := 16#8A43;
   // GBK_TO_UNICODE[28804] := 16#D465;
   // GBK_TO_UNICODE[28805] := 16#8A44;
   // GBK_TO_UNICODE[28806] := 16#D466;
   // GBK_TO_UNICODE[28807] := 16#8A45;
   // GBK_TO_UNICODE[28808] := 16#D467;
   // GBK_TO_UNICODE[28809] := 16#8A46;
   // GBK_TO_UNICODE[28810] := 16#D468;
   // GBK_TO_UNICODE[28811] := 16#8A47;
   // GBK_TO_UNICODE[28812] := 16#D469;
   // GBK_TO_UNICODE[28813] := 16#8A49;
   // GBK_TO_UNICODE[28814] := 16#D46A;
   // GBK_TO_UNICODE[28815] := 16#8A4A;
   // GBK_TO_UNICODE[28816] := 16#D46B;
   // GBK_TO_UNICODE[28817] := 16#8A4B;
   // GBK_TO_UNICODE[28818] := 16#D46C;
   // GBK_TO_UNICODE[28819] := 16#8A4C;
   // GBK_TO_UNICODE[28820] := 16#D46D;
   // GBK_TO_UNICODE[28821] := 16#8A4D;
   // GBK_TO_UNICODE[28822] := 16#D46E;
   // GBK_TO_UNICODE[28823] := 16#8A4E;
   // GBK_TO_UNICODE[28824] := 16#D46F;
   // GBK_TO_UNICODE[28825] := 16#8A4F;
   // GBK_TO_UNICODE[28826] := 16#D470;
   // GBK_TO_UNICODE[28827] := 16#8A50;
   // GBK_TO_UNICODE[28828] := 16#D471;
   // GBK_TO_UNICODE[28829] := 16#8A51;
   // GBK_TO_UNICODE[28830] := 16#D472;
   // GBK_TO_UNICODE[28831] := 16#8A52;
   // GBK_TO_UNICODE[28832] := 16#D473;
   // GBK_TO_UNICODE[28833] := 16#8A53;
   // GBK_TO_UNICODE[28834] := 16#D474;
   // GBK_TO_UNICODE[28835] := 16#8A54;
   // GBK_TO_UNICODE[28836] := 16#D475;
   // GBK_TO_UNICODE[28837] := 16#8A55;
   // GBK_TO_UNICODE[28838] := 16#D476;
   // GBK_TO_UNICODE[28839] := 16#8A56;
   // GBK_TO_UNICODE[28840] := 16#D477;
   // GBK_TO_UNICODE[28841] := 16#8A57;
   // GBK_TO_UNICODE[28842] := 16#D478;
   // GBK_TO_UNICODE[28843] := 16#8A58;
   // GBK_TO_UNICODE[28844] := 16#D479;
   // GBK_TO_UNICODE[28845] := 16#8A59;
   // GBK_TO_UNICODE[28846] := 16#D47A;
   // GBK_TO_UNICODE[28847] := 16#8A5A;
   // GBK_TO_UNICODE[28848] := 16#D47B;
   // GBK_TO_UNICODE[28849] := 16#8A5B;
   // GBK_TO_UNICODE[28850] := 16#D47C;
   // GBK_TO_UNICODE[28851] := 16#8A5C;
   // GBK_TO_UNICODE[28852] := 16#D47D;
   // GBK_TO_UNICODE[28853] := 16#8A5D;
   // GBK_TO_UNICODE[28854] := 16#D47E;
   // GBK_TO_UNICODE[28855] := 16#8A5E;
   // GBK_TO_UNICODE[28856] := 16#D480;
   // GBK_TO_UNICODE[28857] := 16#8A5F;
   // GBK_TO_UNICODE[28858] := 16#D481;
   // GBK_TO_UNICODE[28859] := 16#8A60;
   // GBK_TO_UNICODE[28860] := 16#D482;
   // GBK_TO_UNICODE[28861] := 16#8A61;
   // GBK_TO_UNICODE[28862] := 16#D483;
   // GBK_TO_UNICODE[28863] := 16#8A62;
   // GBK_TO_UNICODE[28864] := 16#D484;
   // GBK_TO_UNICODE[28865] := 16#8A63;
   // GBK_TO_UNICODE[28866] := 16#D485;
   // GBK_TO_UNICODE[28867] := 16#8A64;
   // GBK_TO_UNICODE[28868] := 16#D486;
   // GBK_TO_UNICODE[28869] := 16#8A65;
   // GBK_TO_UNICODE[28870] := 16#D487;
   // GBK_TO_UNICODE[28871] := 16#8A66;
   // GBK_TO_UNICODE[28872] := 16#D488;
   // GBK_TO_UNICODE[28873] := 16#8A67;
   // GBK_TO_UNICODE[28874] := 16#D489;
   // GBK_TO_UNICODE[28875] := 16#8A68;
   // GBK_TO_UNICODE[28876] := 16#D48A;
   // GBK_TO_UNICODE[28877] := 16#8A69;
   // GBK_TO_UNICODE[28878] := 16#D48B;
   // GBK_TO_UNICODE[28879] := 16#8A6A;
   // GBK_TO_UNICODE[28880] := 16#D48C;
   // GBK_TO_UNICODE[28881] := 16#8A6B;
   // GBK_TO_UNICODE[28882] := 16#D48D;
   // GBK_TO_UNICODE[28883] := 16#8A6C;
   // GBK_TO_UNICODE[28884] := 16#D48E;
   // GBK_TO_UNICODE[28885] := 16#8A6D;
   // GBK_TO_UNICODE[28886] := 16#D48F;
   // GBK_TO_UNICODE[28887] := 16#8A6E;
   // GBK_TO_UNICODE[28888] := 16#D490;
   // GBK_TO_UNICODE[28889] := 16#8A6F;
   // GBK_TO_UNICODE[28890] := 16#D491;
   // GBK_TO_UNICODE[28891] := 16#8A70;
   // GBK_TO_UNICODE[28892] := 16#D492;
   // GBK_TO_UNICODE[28893] := 16#8A71;
   // GBK_TO_UNICODE[28894] := 16#D493;
   // GBK_TO_UNICODE[28895] := 16#8A72;
   // GBK_TO_UNICODE[28896] := 16#D494;
   // GBK_TO_UNICODE[28897] := 16#8A73;
   // GBK_TO_UNICODE[28898] := 16#D495;
   // GBK_TO_UNICODE[28899] := 16#8A74;
   // GBK_TO_UNICODE[28900] := 16#D496;
   // GBK_TO_UNICODE[28901] := 16#8A75;
   // GBK_TO_UNICODE[28902] := 16#D497;
   // GBK_TO_UNICODE[28903] := 16#8A76;
   // GBK_TO_UNICODE[28904] := 16#D498;
   // GBK_TO_UNICODE[28905] := 16#8A77;
   // GBK_TO_UNICODE[28906] := 16#D499;
   // GBK_TO_UNICODE[28907] := 16#8A78;
   // GBK_TO_UNICODE[28908] := 16#D49A;
   // GBK_TO_UNICODE[28909] := 16#8A7A;
   // GBK_TO_UNICODE[28910] := 16#D49B;
   // GBK_TO_UNICODE[28911] := 16#8A7B;
   // GBK_TO_UNICODE[28912] := 16#D49C;
   // GBK_TO_UNICODE[28913] := 16#8A7C;
   // GBK_TO_UNICODE[28914] := 16#D49D;
   // GBK_TO_UNICODE[28915] := 16#8A7D;
   // GBK_TO_UNICODE[28916] := 16#D49E;
   // GBK_TO_UNICODE[28917] := 16#8A7E;
   // GBK_TO_UNICODE[28918] := 16#D49F;
   // GBK_TO_UNICODE[28919] := 16#8A7F;
   // GBK_TO_UNICODE[28920] := 16#D4A0;
   // GBK_TO_UNICODE[28921] := 16#8A80;
   // GBK_TO_UNICODE[28922] := 16#D4A1;
   // GBK_TO_UNICODE[28923] := 16#6D74;
   // GBK_TO_UNICODE[28924] := 16#D4A2;
   // GBK_TO_UNICODE[28925] := 16#5BD3;
   // GBK_TO_UNICODE[28926] := 16#D4A3;
   // GBK_TO_UNICODE[28927] := 16#88D5;
   // GBK_TO_UNICODE[28928] := 16#D4A4;
   // GBK_TO_UNICODE[28929] := 16#9884;
   // GBK_TO_UNICODE[28930] := 16#D4A5;
   // GBK_TO_UNICODE[28931] := 16#8C6B;
   // GBK_TO_UNICODE[28932] := 16#D4A6;
   // GBK_TO_UNICODE[28933] := 16#9A6D;
   // GBK_TO_UNICODE[28934] := 16#D4A7;
   // GBK_TO_UNICODE[28935] := 16#9E33;
   // GBK_TO_UNICODE[28936] := 16#D4A8;
   // GBK_TO_UNICODE[28937] := 16#6E0A;
   // GBK_TO_UNICODE[28938] := 16#D4A9;
   // GBK_TO_UNICODE[28939] := 16#51A4;
   // GBK_TO_UNICODE[28940] := 16#D4AA;
   // GBK_TO_UNICODE[28941] := 16#5143;
   // GBK_TO_UNICODE[28942] := 16#D4AB;
   // GBK_TO_UNICODE[28943] := 16#57A3;
   // GBK_TO_UNICODE[28944] := 16#D4AC;
   // GBK_TO_UNICODE[28945] := 16#8881;
   // GBK_TO_UNICODE[28946] := 16#D4AD;
   // GBK_TO_UNICODE[28947] := 16#539F;
   // GBK_TO_UNICODE[28948] := 16#D4AE;
   // GBK_TO_UNICODE[28949] := 16#63F4;
   // GBK_TO_UNICODE[28950] := 16#D4AF;
   // GBK_TO_UNICODE[28951] := 16#8F95;
   // GBK_TO_UNICODE[28952] := 16#D4B0;
   // GBK_TO_UNICODE[28953] := 16#56ED;
   // GBK_TO_UNICODE[28954] := 16#D4B1;
   // GBK_TO_UNICODE[28955] := 16#5458;
   // GBK_TO_UNICODE[28956] := 16#D4B2;
   // GBK_TO_UNICODE[28957] := 16#5706;
   // GBK_TO_UNICODE[28958] := 16#D4B3;
   // GBK_TO_UNICODE[28959] := 16#733F;
   // GBK_TO_UNICODE[28960] := 16#D4B4;
   // GBK_TO_UNICODE[28961] := 16#6E90;
   // GBK_TO_UNICODE[28962] := 16#D4B5;
   // GBK_TO_UNICODE[28963] := 16#7F18;
   // GBK_TO_UNICODE[28964] := 16#D4B6;
   // GBK_TO_UNICODE[28965] := 16#8FDC;
   // GBK_TO_UNICODE[28966] := 16#D4B7;
   // GBK_TO_UNICODE[28967] := 16#82D1;
   // GBK_TO_UNICODE[28968] := 16#D4B8;
   // GBK_TO_UNICODE[28969] := 16#613F;
   // GBK_TO_UNICODE[28970] := 16#D4B9;
   // GBK_TO_UNICODE[28971] := 16#6028;
   // GBK_TO_UNICODE[28972] := 16#D4BA;
   // GBK_TO_UNICODE[28973] := 16#9662;
   // GBK_TO_UNICODE[28974] := 16#D4BB;
   // GBK_TO_UNICODE[28975] := 16#66F0;
   // GBK_TO_UNICODE[28976] := 16#D4BC;
   // GBK_TO_UNICODE[28977] := 16#7EA6;
   // GBK_TO_UNICODE[28978] := 16#D4BD;
   // GBK_TO_UNICODE[28979] := 16#8D8A;
   // GBK_TO_UNICODE[28980] := 16#D4BE;
   // GBK_TO_UNICODE[28981] := 16#8DC3;
   // GBK_TO_UNICODE[28982] := 16#D4BF;
   // GBK_TO_UNICODE[28983] := 16#94A5;
   // GBK_TO_UNICODE[28984] := 16#D4C0;
   // GBK_TO_UNICODE[28985] := 16#5CB3;
   // GBK_TO_UNICODE[28986] := 16#D4C1;
   // GBK_TO_UNICODE[28987] := 16#7CA4;
   // GBK_TO_UNICODE[28988] := 16#D4C2;
   // GBK_TO_UNICODE[28989] := 16#6708;
   // GBK_TO_UNICODE[28990] := 16#D4C3;
   // GBK_TO_UNICODE[28991] := 16#60A6;
   // GBK_TO_UNICODE[28992] := 16#D4C4;
   // GBK_TO_UNICODE[28993] := 16#9605;
   // GBK_TO_UNICODE[28994] := 16#D4C5;
   // GBK_TO_UNICODE[28995] := 16#8018;
   // GBK_TO_UNICODE[28996] := 16#D4C6;
   // GBK_TO_UNICODE[28997] := 16#4E91;
   // GBK_TO_UNICODE[28998] := 16#D4C7;
   // GBK_TO_UNICODE[28999] := 16#90E7;
   // GBK_TO_UNICODE[29000] := 16#D4C8;
   // GBK_TO_UNICODE[29001] := 16#5300;
   // GBK_TO_UNICODE[29002] := 16#D4C9;
   // GBK_TO_UNICODE[29003] := 16#9668;
   // GBK_TO_UNICODE[29004] := 16#D4CA;
   // GBK_TO_UNICODE[29005] := 16#5141;
   // GBK_TO_UNICODE[29006] := 16#D4CB;
   // GBK_TO_UNICODE[29007] := 16#8FD0;
   // GBK_TO_UNICODE[29008] := 16#D4CC;
   // GBK_TO_UNICODE[29009] := 16#8574;
   // GBK_TO_UNICODE[29010] := 16#D4CD;
   // GBK_TO_UNICODE[29011] := 16#915D;
   // GBK_TO_UNICODE[29012] := 16#D4CE;
   // GBK_TO_UNICODE[29013] := 16#6655;
   // GBK_TO_UNICODE[29014] := 16#D4CF;
   // GBK_TO_UNICODE[29015] := 16#97F5;
   // GBK_TO_UNICODE[29016] := 16#D4D0;
   // GBK_TO_UNICODE[29017] := 16#5B55;
   // GBK_TO_UNICODE[29018] := 16#D4D1;
   // GBK_TO_UNICODE[29019] := 16#531D;
   // GBK_TO_UNICODE[29020] := 16#D4D2;
   // GBK_TO_UNICODE[29021] := 16#7838;
   // GBK_TO_UNICODE[29022] := 16#D4D3;
   // GBK_TO_UNICODE[29023] := 16#6742;
   // GBK_TO_UNICODE[29024] := 16#D4D4;
   // GBK_TO_UNICODE[29025] := 16#683D;
   // GBK_TO_UNICODE[29026] := 16#D4D5;
   // GBK_TO_UNICODE[29027] := 16#54C9;
   // GBK_TO_UNICODE[29028] := 16#D4D6;
   // GBK_TO_UNICODE[29029] := 16#707E;
   // GBK_TO_UNICODE[29030] := 16#D4D7;
   // GBK_TO_UNICODE[29031] := 16#5BB0;
   // GBK_TO_UNICODE[29032] := 16#D4D8;
   // GBK_TO_UNICODE[29033] := 16#8F7D;
   // GBK_TO_UNICODE[29034] := 16#D4D9;
   // GBK_TO_UNICODE[29035] := 16#518D;
   // GBK_TO_UNICODE[29036] := 16#D4DA;
   // GBK_TO_UNICODE[29037] := 16#5728;
   // GBK_TO_UNICODE[29038] := 16#D4DB;
   // GBK_TO_UNICODE[29039] := 16#54B1;
   // GBK_TO_UNICODE[29040] := 16#D4DC;
   // GBK_TO_UNICODE[29041] := 16#6512;
   // GBK_TO_UNICODE[29042] := 16#D4DD;
   // GBK_TO_UNICODE[29043] := 16#6682;
   // GBK_TO_UNICODE[29044] := 16#D4DE;
   // GBK_TO_UNICODE[29045] := 16#8D5E;
   // GBK_TO_UNICODE[29046] := 16#D4DF;
   // GBK_TO_UNICODE[29047] := 16#8D43;
   // GBK_TO_UNICODE[29048] := 16#D4E0;
   // GBK_TO_UNICODE[29049] := 16#810F;
   // GBK_TO_UNICODE[29050] := 16#D4E1;
   // GBK_TO_UNICODE[29051] := 16#846C;
   // GBK_TO_UNICODE[29052] := 16#D4E2;
   // GBK_TO_UNICODE[29053] := 16#906D;
   // GBK_TO_UNICODE[29054] := 16#D4E3;
   // GBK_TO_UNICODE[29055] := 16#7CDF;
   // GBK_TO_UNICODE[29056] := 16#D4E4;
   // GBK_TO_UNICODE[29057] := 16#51FF;
   // GBK_TO_UNICODE[29058] := 16#D4E5;
   // GBK_TO_UNICODE[29059] := 16#85FB;
   // GBK_TO_UNICODE[29060] := 16#D4E6;
   // GBK_TO_UNICODE[29061] := 16#67A3;
   // GBK_TO_UNICODE[29062] := 16#D4E7;
   // GBK_TO_UNICODE[29063] := 16#65E9;
   // GBK_TO_UNICODE[29064] := 16#D4E8;
   // GBK_TO_UNICODE[29065] := 16#6FA1;
   // GBK_TO_UNICODE[29066] := 16#D4E9;
   // GBK_TO_UNICODE[29067] := 16#86A4;
   // GBK_TO_UNICODE[29068] := 16#D4EA;
   // GBK_TO_UNICODE[29069] := 16#8E81;
   // GBK_TO_UNICODE[29070] := 16#D4EB;
   // GBK_TO_UNICODE[29071] := 16#566A;
   // GBK_TO_UNICODE[29072] := 16#D4EC;
   // GBK_TO_UNICODE[29073] := 16#9020;
   // GBK_TO_UNICODE[29074] := 16#D4ED;
   // GBK_TO_UNICODE[29075] := 16#7682;
   // GBK_TO_UNICODE[29076] := 16#D4EE;
   // GBK_TO_UNICODE[29077] := 16#7076;
   // GBK_TO_UNICODE[29078] := 16#D4EF;
   // GBK_TO_UNICODE[29079] := 16#71E5;
   // GBK_TO_UNICODE[29080] := 16#D4F0;
   // GBK_TO_UNICODE[29081] := 16#8D23;
   // GBK_TO_UNICODE[29082] := 16#D4F1;
   // GBK_TO_UNICODE[29083] := 16#62E9;
   // GBK_TO_UNICODE[29084] := 16#D4F2;
   // GBK_TO_UNICODE[29085] := 16#5219;
   // GBK_TO_UNICODE[29086] := 16#D4F3;
   // GBK_TO_UNICODE[29087] := 16#6CFD;
   // GBK_TO_UNICODE[29088] := 16#D4F4;
   // GBK_TO_UNICODE[29089] := 16#8D3C;
   // GBK_TO_UNICODE[29090] := 16#D4F5;
   // GBK_TO_UNICODE[29091] := 16#600E;
   // GBK_TO_UNICODE[29092] := 16#D4F6;
   // GBK_TO_UNICODE[29093] := 16#589E;
   // GBK_TO_UNICODE[29094] := 16#D4F7;
   // GBK_TO_UNICODE[29095] := 16#618E;
   // GBK_TO_UNICODE[29096] := 16#D4F8;
   // GBK_TO_UNICODE[29097] := 16#66FE;
   // GBK_TO_UNICODE[29098] := 16#D4F9;
   // GBK_TO_UNICODE[29099] := 16#8D60;
   // GBK_TO_UNICODE[29100] := 16#D4FA;
   // GBK_TO_UNICODE[29101] := 16#624E;
   // GBK_TO_UNICODE[29102] := 16#D4FB;
   // GBK_TO_UNICODE[29103] := 16#55B3;
   // GBK_TO_UNICODE[29104] := 16#D4FC;
   // GBK_TO_UNICODE[29105] := 16#6E23;
   // GBK_TO_UNICODE[29106] := 16#D4FD;
   // GBK_TO_UNICODE[29107] := 16#672D;
   // GBK_TO_UNICODE[29108] := 16#D4FE;
   // GBK_TO_UNICODE[29109] := 16#8F67;
   // GBK_TO_UNICODE[29110] := 16#D540;
   // GBK_TO_UNICODE[29111] := 16#8A81;
   // GBK_TO_UNICODE[29112] := 16#D541;
   // GBK_TO_UNICODE[29113] := 16#8A82;
   // GBK_TO_UNICODE[29114] := 16#D542;
   // GBK_TO_UNICODE[29115] := 16#8A83;
   // GBK_TO_UNICODE[29116] := 16#D543;
   // GBK_TO_UNICODE[29117] := 16#8A84;
   // GBK_TO_UNICODE[29118] := 16#D544;
   // GBK_TO_UNICODE[29119] := 16#8A85;
   // GBK_TO_UNICODE[29120] := 16#D545;
   // GBK_TO_UNICODE[29121] := 16#8A86;
   // GBK_TO_UNICODE[29122] := 16#D546;
   // GBK_TO_UNICODE[29123] := 16#8A87;
   // GBK_TO_UNICODE[29124] := 16#D547;
   // GBK_TO_UNICODE[29125] := 16#8A88;
   // GBK_TO_UNICODE[29126] := 16#D548;
   // GBK_TO_UNICODE[29127] := 16#8A8B;
   // GBK_TO_UNICODE[29128] := 16#D549;
   // GBK_TO_UNICODE[29129] := 16#8A8C;
   // GBK_TO_UNICODE[29130] := 16#D54A;
   // GBK_TO_UNICODE[29131] := 16#8A8D;
   // GBK_TO_UNICODE[29132] := 16#D54B;
   // GBK_TO_UNICODE[29133] := 16#8A8E;
   // GBK_TO_UNICODE[29134] := 16#D54C;
   // GBK_TO_UNICODE[29135] := 16#8A8F;
   // GBK_TO_UNICODE[29136] := 16#D54D;
   // GBK_TO_UNICODE[29137] := 16#8A90;
   // GBK_TO_UNICODE[29138] := 16#D54E;
   // GBK_TO_UNICODE[29139] := 16#8A91;
   // GBK_TO_UNICODE[29140] := 16#D54F;
   // GBK_TO_UNICODE[29141] := 16#8A92;
   // GBK_TO_UNICODE[29142] := 16#D550;
   // GBK_TO_UNICODE[29143] := 16#8A94;
   // GBK_TO_UNICODE[29144] := 16#D551;
   // GBK_TO_UNICODE[29145] := 16#8A95;
   // GBK_TO_UNICODE[29146] := 16#D552;
   // GBK_TO_UNICODE[29147] := 16#8A96;
   // GBK_TO_UNICODE[29148] := 16#D553;
   // GBK_TO_UNICODE[29149] := 16#8A97;
   // GBK_TO_UNICODE[29150] := 16#D554;
   // GBK_TO_UNICODE[29151] := 16#8A98;
   // GBK_TO_UNICODE[29152] := 16#D555;
   // GBK_TO_UNICODE[29153] := 16#8A99;
   // GBK_TO_UNICODE[29154] := 16#D556;
   // GBK_TO_UNICODE[29155] := 16#8A9A;
   // GBK_TO_UNICODE[29156] := 16#D557;
   // GBK_TO_UNICODE[29157] := 16#8A9B;
   // GBK_TO_UNICODE[29158] := 16#D558;
   // GBK_TO_UNICODE[29159] := 16#8A9C;
   // GBK_TO_UNICODE[29160] := 16#D559;
   // GBK_TO_UNICODE[29161] := 16#8A9D;
   // GBK_TO_UNICODE[29162] := 16#D55A;
   // GBK_TO_UNICODE[29163] := 16#8A9E;
   // GBK_TO_UNICODE[29164] := 16#D55B;
   // GBK_TO_UNICODE[29165] := 16#8A9F;
   // GBK_TO_UNICODE[29166] := 16#D55C;
   // GBK_TO_UNICODE[29167] := 16#8AA0;
   // GBK_TO_UNICODE[29168] := 16#D55D;
   // GBK_TO_UNICODE[29169] := 16#8AA1;
   // GBK_TO_UNICODE[29170] := 16#D55E;
   // GBK_TO_UNICODE[29171] := 16#8AA2;
   // GBK_TO_UNICODE[29172] := 16#D55F;
   // GBK_TO_UNICODE[29173] := 16#8AA3;
   // GBK_TO_UNICODE[29174] := 16#D560;
   // GBK_TO_UNICODE[29175] := 16#8AA4;
   // GBK_TO_UNICODE[29176] := 16#D561;
   // GBK_TO_UNICODE[29177] := 16#8AA5;
   // GBK_TO_UNICODE[29178] := 16#D562;
   // GBK_TO_UNICODE[29179] := 16#8AA6;
   // GBK_TO_UNICODE[29180] := 16#D563;
   // GBK_TO_UNICODE[29181] := 16#8AA7;
   // GBK_TO_UNICODE[29182] := 16#D564;
   // GBK_TO_UNICODE[29183] := 16#8AA8;
   // GBK_TO_UNICODE[29184] := 16#D565;
   // GBK_TO_UNICODE[29185] := 16#8AA9;
   // GBK_TO_UNICODE[29186] := 16#D566;
   // GBK_TO_UNICODE[29187] := 16#8AAA;
   // GBK_TO_UNICODE[29188] := 16#D567;
   // GBK_TO_UNICODE[29189] := 16#8AAB;
   // GBK_TO_UNICODE[29190] := 16#D568;
   // GBK_TO_UNICODE[29191] := 16#8AAC;
   // GBK_TO_UNICODE[29192] := 16#D569;
   // GBK_TO_UNICODE[29193] := 16#8AAD;
   // GBK_TO_UNICODE[29194] := 16#D56A;
   // GBK_TO_UNICODE[29195] := 16#8AAE;
   // GBK_TO_UNICODE[29196] := 16#D56B;
   // GBK_TO_UNICODE[29197] := 16#8AAF;
   // GBK_TO_UNICODE[29198] := 16#D56C;
   // GBK_TO_UNICODE[29199] := 16#8AB0;
   // GBK_TO_UNICODE[29200] := 16#D56D;
   // GBK_TO_UNICODE[29201] := 16#8AB1;
   // GBK_TO_UNICODE[29202] := 16#D56E;
   // GBK_TO_UNICODE[29203] := 16#8AB2;
   // GBK_TO_UNICODE[29204] := 16#D56F;
   // GBK_TO_UNICODE[29205] := 16#8AB3;
   // GBK_TO_UNICODE[29206] := 16#D570;
   // GBK_TO_UNICODE[29207] := 16#8AB4;
   // GBK_TO_UNICODE[29208] := 16#D571;
   // GBK_TO_UNICODE[29209] := 16#8AB5;
   // GBK_TO_UNICODE[29210] := 16#D572;
   // GBK_TO_UNICODE[29211] := 16#8AB6;
   // GBK_TO_UNICODE[29212] := 16#D573;
   // GBK_TO_UNICODE[29213] := 16#8AB7;
   // GBK_TO_UNICODE[29214] := 16#D574;
   // GBK_TO_UNICODE[29215] := 16#8AB8;
   // GBK_TO_UNICODE[29216] := 16#D575;
   // GBK_TO_UNICODE[29217] := 16#8AB9;
   // GBK_TO_UNICODE[29218] := 16#D576;
   // GBK_TO_UNICODE[29219] := 16#8ABA;
   // GBK_TO_UNICODE[29220] := 16#D577;
   // GBK_TO_UNICODE[29221] := 16#8ABB;
   // GBK_TO_UNICODE[29222] := 16#D578;
   // GBK_TO_UNICODE[29223] := 16#8ABC;
   // GBK_TO_UNICODE[29224] := 16#D579;
   // GBK_TO_UNICODE[29225] := 16#8ABD;
   // GBK_TO_UNICODE[29226] := 16#D57A;
   // GBK_TO_UNICODE[29227] := 16#8ABE;
   // GBK_TO_UNICODE[29228] := 16#D57B;
   // GBK_TO_UNICODE[29229] := 16#8ABF;
   // GBK_TO_UNICODE[29230] := 16#D57C;
   // GBK_TO_UNICODE[29231] := 16#8AC0;
   // GBK_TO_UNICODE[29232] := 16#D57D;
   // GBK_TO_UNICODE[29233] := 16#8AC1;
   // GBK_TO_UNICODE[29234] := 16#D57E;
   // GBK_TO_UNICODE[29235] := 16#8AC2;
   // GBK_TO_UNICODE[29236] := 16#D580;
   // GBK_TO_UNICODE[29237] := 16#8AC3;
   // GBK_TO_UNICODE[29238] := 16#D581;
   // GBK_TO_UNICODE[29239] := 16#8AC4;
   // GBK_TO_UNICODE[29240] := 16#D582;
   // GBK_TO_UNICODE[29241] := 16#8AC5;
   // GBK_TO_UNICODE[29242] := 16#D583;
   // GBK_TO_UNICODE[29243] := 16#8AC6;
   // GBK_TO_UNICODE[29244] := 16#D584;
   // GBK_TO_UNICODE[29245] := 16#8AC7;
   // GBK_TO_UNICODE[29246] := 16#D585;
   // GBK_TO_UNICODE[29247] := 16#8AC8;
   // GBK_TO_UNICODE[29248] := 16#D586;
   // GBK_TO_UNICODE[29249] := 16#8AC9;
   // GBK_TO_UNICODE[29250] := 16#D587;
   // GBK_TO_UNICODE[29251] := 16#8ACA;
   // GBK_TO_UNICODE[29252] := 16#D588;
   // GBK_TO_UNICODE[29253] := 16#8ACB;
   // GBK_TO_UNICODE[29254] := 16#D589;
   // GBK_TO_UNICODE[29255] := 16#8ACC;
   // GBK_TO_UNICODE[29256] := 16#D58A;
   // GBK_TO_UNICODE[29257] := 16#8ACD;
   // GBK_TO_UNICODE[29258] := 16#D58B;
   // GBK_TO_UNICODE[29259] := 16#8ACE;
   // GBK_TO_UNICODE[29260] := 16#D58C;
   // GBK_TO_UNICODE[29261] := 16#8ACF;
   // GBK_TO_UNICODE[29262] := 16#D58D;
   // GBK_TO_UNICODE[29263] := 16#8AD0;
   // GBK_TO_UNICODE[29264] := 16#D58E;
   // GBK_TO_UNICODE[29265] := 16#8AD1;
   // GBK_TO_UNICODE[29266] := 16#D58F;
   // GBK_TO_UNICODE[29267] := 16#8AD2;
   // GBK_TO_UNICODE[29268] := 16#D590;
   // GBK_TO_UNICODE[29269] := 16#8AD3;
   // GBK_TO_UNICODE[29270] := 16#D591;
   // GBK_TO_UNICODE[29271] := 16#8AD4;
   // GBK_TO_UNICODE[29272] := 16#D592;
   // GBK_TO_UNICODE[29273] := 16#8AD5;
   // GBK_TO_UNICODE[29274] := 16#D593;
   // GBK_TO_UNICODE[29275] := 16#8AD6;
   // GBK_TO_UNICODE[29276] := 16#D594;
   // GBK_TO_UNICODE[29277] := 16#8AD7;
   // GBK_TO_UNICODE[29278] := 16#D595;
   // GBK_TO_UNICODE[29279] := 16#8AD8;
   // GBK_TO_UNICODE[29280] := 16#D596;
   // GBK_TO_UNICODE[29281] := 16#8AD9;
   // GBK_TO_UNICODE[29282] := 16#D597;
   // GBK_TO_UNICODE[29283] := 16#8ADA;
   // GBK_TO_UNICODE[29284] := 16#D598;
   // GBK_TO_UNICODE[29285] := 16#8ADB;
   // GBK_TO_UNICODE[29286] := 16#D599;
   // GBK_TO_UNICODE[29287] := 16#8ADC;
   // GBK_TO_UNICODE[29288] := 16#D59A;
   // GBK_TO_UNICODE[29289] := 16#8ADD;
   // GBK_TO_UNICODE[29290] := 16#D59B;
   // GBK_TO_UNICODE[29291] := 16#8ADE;
   // GBK_TO_UNICODE[29292] := 16#D59C;
   // GBK_TO_UNICODE[29293] := 16#8ADF;
   // GBK_TO_UNICODE[29294] := 16#D59D;
   // GBK_TO_UNICODE[29295] := 16#8AE0;
   // GBK_TO_UNICODE[29296] := 16#D59E;
   // GBK_TO_UNICODE[29297] := 16#8AE1;
   // GBK_TO_UNICODE[29298] := 16#D59F;
   // GBK_TO_UNICODE[29299] := 16#8AE2;
   // GBK_TO_UNICODE[29300] := 16#D5A0;
   // GBK_TO_UNICODE[29301] := 16#8AE3;
   // GBK_TO_UNICODE[29302] := 16#D5A1;
   // GBK_TO_UNICODE[29303] := 16#94E1;
   // GBK_TO_UNICODE[29304] := 16#D5A2;
   // GBK_TO_UNICODE[29305] := 16#95F8;
   // GBK_TO_UNICODE[29306] := 16#D5A3;
   // GBK_TO_UNICODE[29307] := 16#7728;
   // GBK_TO_UNICODE[29308] := 16#D5A4;
   // GBK_TO_UNICODE[29309] := 16#6805;
   // GBK_TO_UNICODE[29310] := 16#D5A5;
   // GBK_TO_UNICODE[29311] := 16#69A8;
   // GBK_TO_UNICODE[29312] := 16#D5A6;
   // GBK_TO_UNICODE[29313] := 16#548B;
   // GBK_TO_UNICODE[29314] := 16#D5A7;
   // GBK_TO_UNICODE[29315] := 16#4E4D;
   // GBK_TO_UNICODE[29316] := 16#D5A8;
   // GBK_TO_UNICODE[29317] := 16#70B8;
   // GBK_TO_UNICODE[29318] := 16#D5A9;
   // GBK_TO_UNICODE[29319] := 16#8BC8;
   // GBK_TO_UNICODE[29320] := 16#D5AA;
   // GBK_TO_UNICODE[29321] := 16#6458;
   // GBK_TO_UNICODE[29322] := 16#D5AB;
   // GBK_TO_UNICODE[29323] := 16#658B;
   // GBK_TO_UNICODE[29324] := 16#D5AC;
   // GBK_TO_UNICODE[29325] := 16#5B85;
   // GBK_TO_UNICODE[29326] := 16#D5AD;
   // GBK_TO_UNICODE[29327] := 16#7A84;
   // GBK_TO_UNICODE[29328] := 16#D5AE;
   // GBK_TO_UNICODE[29329] := 16#503A;
   // GBK_TO_UNICODE[29330] := 16#D5AF;
   // GBK_TO_UNICODE[29331] := 16#5BE8;
   // GBK_TO_UNICODE[29332] := 16#D5B0;
   // GBK_TO_UNICODE[29333] := 16#77BB;
   // GBK_TO_UNICODE[29334] := 16#D5B1;
   // GBK_TO_UNICODE[29335] := 16#6BE1;
   // GBK_TO_UNICODE[29336] := 16#D5B2;
   // GBK_TO_UNICODE[29337] := 16#8A79;
   // GBK_TO_UNICODE[29338] := 16#D5B3;
   // GBK_TO_UNICODE[29339] := 16#7C98;
   // GBK_TO_UNICODE[29340] := 16#D5B4;
   // GBK_TO_UNICODE[29341] := 16#6CBE;
   // GBK_TO_UNICODE[29342] := 16#D5B5;
   // GBK_TO_UNICODE[29343] := 16#76CF;
   // GBK_TO_UNICODE[29344] := 16#D5B6;
   // GBK_TO_UNICODE[29345] := 16#65A9;
   // GBK_TO_UNICODE[29346] := 16#D5B7;
   // GBK_TO_UNICODE[29347] := 16#8F97;
   // GBK_TO_UNICODE[29348] := 16#D5B8;
   // GBK_TO_UNICODE[29349] := 16#5D2D;
   // GBK_TO_UNICODE[29350] := 16#D5B9;
   // GBK_TO_UNICODE[29351] := 16#5C55;
   // GBK_TO_UNICODE[29352] := 16#D5BA;
   // GBK_TO_UNICODE[29353] := 16#8638;
   // GBK_TO_UNICODE[29354] := 16#D5BB;
   // GBK_TO_UNICODE[29355] := 16#6808;
   // GBK_TO_UNICODE[29356] := 16#D5BC;
   // GBK_TO_UNICODE[29357] := 16#5360;
   // GBK_TO_UNICODE[29358] := 16#D5BD;
   // GBK_TO_UNICODE[29359] := 16#6218;
   // GBK_TO_UNICODE[29360] := 16#D5BE;
   // GBK_TO_UNICODE[29361] := 16#7AD9;
   // GBK_TO_UNICODE[29362] := 16#D5BF;
   // GBK_TO_UNICODE[29363] := 16#6E5B;
   // GBK_TO_UNICODE[29364] := 16#D5C0;
   // GBK_TO_UNICODE[29365] := 16#7EFD;
   // GBK_TO_UNICODE[29366] := 16#D5C1;
   // GBK_TO_UNICODE[29367] := 16#6A1F;
   // GBK_TO_UNICODE[29368] := 16#D5C2;
   // GBK_TO_UNICODE[29369] := 16#7AE0;
   // GBK_TO_UNICODE[29370] := 16#D5C3;
   // GBK_TO_UNICODE[29371] := 16#5F70;
   // GBK_TO_UNICODE[29372] := 16#D5C4;
   // GBK_TO_UNICODE[29373] := 16#6F33;
   // GBK_TO_UNICODE[29374] := 16#D5C5;
   // GBK_TO_UNICODE[29375] := 16#5F20;
   // GBK_TO_UNICODE[29376] := 16#D5C6;
   // GBK_TO_UNICODE[29377] := 16#638C;
   // GBK_TO_UNICODE[29378] := 16#D5C7;
   // GBK_TO_UNICODE[29379] := 16#6DA8;
   // GBK_TO_UNICODE[29380] := 16#D5C8;
   // GBK_TO_UNICODE[29381] := 16#6756;
   // GBK_TO_UNICODE[29382] := 16#D5C9;
   // GBK_TO_UNICODE[29383] := 16#4E08;
   // GBK_TO_UNICODE[29384] := 16#D5CA;
   // GBK_TO_UNICODE[29385] := 16#5E10;
   // GBK_TO_UNICODE[29386] := 16#D5CB;
   // GBK_TO_UNICODE[29387] := 16#8D26;
   // GBK_TO_UNICODE[29388] := 16#D5CC;
   // GBK_TO_UNICODE[29389] := 16#4ED7;
   // GBK_TO_UNICODE[29390] := 16#D5CD;
   // GBK_TO_UNICODE[29391] := 16#80C0;
   // GBK_TO_UNICODE[29392] := 16#D5CE;
   // GBK_TO_UNICODE[29393] := 16#7634;
   // GBK_TO_UNICODE[29394] := 16#D5CF;
   // GBK_TO_UNICODE[29395] := 16#969C;
   // GBK_TO_UNICODE[29396] := 16#D5D0;
   // GBK_TO_UNICODE[29397] := 16#62DB;
   // GBK_TO_UNICODE[29398] := 16#D5D1;
   // GBK_TO_UNICODE[29399] := 16#662D;
   // GBK_TO_UNICODE[29400] := 16#D5D2;
   // GBK_TO_UNICODE[29401] := 16#627E;
   // GBK_TO_UNICODE[29402] := 16#D5D3;
   // GBK_TO_UNICODE[29403] := 16#6CBC;
   // GBK_TO_UNICODE[29404] := 16#D5D4;
   // GBK_TO_UNICODE[29405] := 16#8D75;
   // GBK_TO_UNICODE[29406] := 16#D5D5;
   // GBK_TO_UNICODE[29407] := 16#7167;
   // GBK_TO_UNICODE[29408] := 16#D5D6;
   // GBK_TO_UNICODE[29409] := 16#7F69;
   // GBK_TO_UNICODE[29410] := 16#D5D7;
   // GBK_TO_UNICODE[29411] := 16#5146;
   // GBK_TO_UNICODE[29412] := 16#D5D8;
   // GBK_TO_UNICODE[29413] := 16#8087;
   // GBK_TO_UNICODE[29414] := 16#D5D9;
   // GBK_TO_UNICODE[29415] := 16#53EC;
   // GBK_TO_UNICODE[29416] := 16#D5DA;
   // GBK_TO_UNICODE[29417] := 16#906E;
   // GBK_TO_UNICODE[29418] := 16#D5DB;
   // GBK_TO_UNICODE[29419] := 16#6298;
   // GBK_TO_UNICODE[29420] := 16#D5DC;
   // GBK_TO_UNICODE[29421] := 16#54F2;
   // GBK_TO_UNICODE[29422] := 16#D5DD;
   // GBK_TO_UNICODE[29423] := 16#86F0;
   // GBK_TO_UNICODE[29424] := 16#D5DE;
   // GBK_TO_UNICODE[29425] := 16#8F99;
   // GBK_TO_UNICODE[29426] := 16#D5DF;
   // GBK_TO_UNICODE[29427] := 16#8005;
   // GBK_TO_UNICODE[29428] := 16#D5E0;
   // GBK_TO_UNICODE[29429] := 16#9517;
   // GBK_TO_UNICODE[29430] := 16#D5E1;
   // GBK_TO_UNICODE[29431] := 16#8517;
   // GBK_TO_UNICODE[29432] := 16#D5E2;
   // GBK_TO_UNICODE[29433] := 16#8FD9;
   // GBK_TO_UNICODE[29434] := 16#D5E3;
   // GBK_TO_UNICODE[29435] := 16#6D59;
   // GBK_TO_UNICODE[29436] := 16#D5E4;
   // GBK_TO_UNICODE[29437] := 16#73CD;
   // GBK_TO_UNICODE[29438] := 16#D5E5;
   // GBK_TO_UNICODE[29439] := 16#659F;
   // GBK_TO_UNICODE[29440] := 16#D5E6;
   // GBK_TO_UNICODE[29441] := 16#771F;
   // GBK_TO_UNICODE[29442] := 16#D5E7;
   // GBK_TO_UNICODE[29443] := 16#7504;
   // GBK_TO_UNICODE[29444] := 16#D5E8;
   // GBK_TO_UNICODE[29445] := 16#7827;
   // GBK_TO_UNICODE[29446] := 16#D5E9;
   // GBK_TO_UNICODE[29447] := 16#81FB;
   // GBK_TO_UNICODE[29448] := 16#D5EA;
   // GBK_TO_UNICODE[29449] := 16#8D1E;
   // GBK_TO_UNICODE[29450] := 16#D5EB;
   // GBK_TO_UNICODE[29451] := 16#9488;
   // GBK_TO_UNICODE[29452] := 16#D5EC;
   // GBK_TO_UNICODE[29453] := 16#4FA6;
   // GBK_TO_UNICODE[29454] := 16#D5ED;
   // GBK_TO_UNICODE[29455] := 16#6795;
   // GBK_TO_UNICODE[29456] := 16#D5EE;
   // GBK_TO_UNICODE[29457] := 16#75B9;
   // GBK_TO_UNICODE[29458] := 16#D5EF;
   // GBK_TO_UNICODE[29459] := 16#8BCA;
   // GBK_TO_UNICODE[29460] := 16#D5F0;
   // GBK_TO_UNICODE[29461] := 16#9707;
   // GBK_TO_UNICODE[29462] := 16#D5F1;
   // GBK_TO_UNICODE[29463] := 16#632F;
   // GBK_TO_UNICODE[29464] := 16#D5F2;
   // GBK_TO_UNICODE[29465] := 16#9547;
   // GBK_TO_UNICODE[29466] := 16#D5F3;
   // GBK_TO_UNICODE[29467] := 16#9635;
   // GBK_TO_UNICODE[29468] := 16#D5F4;
   // GBK_TO_UNICODE[29469] := 16#84B8;
   // GBK_TO_UNICODE[29470] := 16#D5F5;
   // GBK_TO_UNICODE[29471] := 16#6323;
   // GBK_TO_UNICODE[29472] := 16#D5F6;
   // GBK_TO_UNICODE[29473] := 16#7741;
   // GBK_TO_UNICODE[29474] := 16#D5F7;
   // GBK_TO_UNICODE[29475] := 16#5F81;
   // GBK_TO_UNICODE[29476] := 16#D5F8;
   // GBK_TO_UNICODE[29477] := 16#72F0;
   // GBK_TO_UNICODE[29478] := 16#D5F9;
   // GBK_TO_UNICODE[29479] := 16#4E89;
   // GBK_TO_UNICODE[29480] := 16#D5FA;
   // GBK_TO_UNICODE[29481] := 16#6014;
   // GBK_TO_UNICODE[29482] := 16#D5FB;
   // GBK_TO_UNICODE[29483] := 16#6574;
   // GBK_TO_UNICODE[29484] := 16#D5FC;
   // GBK_TO_UNICODE[29485] := 16#62EF;
   // GBK_TO_UNICODE[29486] := 16#D5FD;
   // GBK_TO_UNICODE[29487] := 16#6B63;
   // GBK_TO_UNICODE[29488] := 16#D5FE;
   // GBK_TO_UNICODE[29489] := 16#653F;
   // GBK_TO_UNICODE[29490] := 16#D640;
   // GBK_TO_UNICODE[29491] := 16#8AE4;
   // GBK_TO_UNICODE[29492] := 16#D641;
   // GBK_TO_UNICODE[29493] := 16#8AE5;
   // GBK_TO_UNICODE[29494] := 16#D642;
   // GBK_TO_UNICODE[29495] := 16#8AE6;
   // GBK_TO_UNICODE[29496] := 16#D643;
   // GBK_TO_UNICODE[29497] := 16#8AE7;
   // GBK_TO_UNICODE[29498] := 16#D644;
   // GBK_TO_UNICODE[29499] := 16#8AE8;
   // GBK_TO_UNICODE[29500] := 16#D645;
   // GBK_TO_UNICODE[29501] := 16#8AE9;
   // GBK_TO_UNICODE[29502] := 16#D646;
   // GBK_TO_UNICODE[29503] := 16#8AEA;
   // GBK_TO_UNICODE[29504] := 16#D647;
   // GBK_TO_UNICODE[29505] := 16#8AEB;
   // GBK_TO_UNICODE[29506] := 16#D648;
   // GBK_TO_UNICODE[29507] := 16#8AEC;
   // GBK_TO_UNICODE[29508] := 16#D649;
   // GBK_TO_UNICODE[29509] := 16#8AED;
   // GBK_TO_UNICODE[29510] := 16#D64A;
   // GBK_TO_UNICODE[29511] := 16#8AEE;
   // GBK_TO_UNICODE[29512] := 16#D64B;
   // GBK_TO_UNICODE[29513] := 16#8AEF;
   // GBK_TO_UNICODE[29514] := 16#D64C;
   // GBK_TO_UNICODE[29515] := 16#8AF0;
   // GBK_TO_UNICODE[29516] := 16#D64D;
   // GBK_TO_UNICODE[29517] := 16#8AF1;
   // GBK_TO_UNICODE[29518] := 16#D64E;
   // GBK_TO_UNICODE[29519] := 16#8AF2;
   // GBK_TO_UNICODE[29520] := 16#D64F;
   // GBK_TO_UNICODE[29521] := 16#8AF3;
   // GBK_TO_UNICODE[29522] := 16#D650;
   // GBK_TO_UNICODE[29523] := 16#8AF4;
   // GBK_TO_UNICODE[29524] := 16#D651;
   // GBK_TO_UNICODE[29525] := 16#8AF5;
   // GBK_TO_UNICODE[29526] := 16#D652;
   // GBK_TO_UNICODE[29527] := 16#8AF6;
   // GBK_TO_UNICODE[29528] := 16#D653;
   // GBK_TO_UNICODE[29529] := 16#8AF7;
   // GBK_TO_UNICODE[29530] := 16#D654;
   // GBK_TO_UNICODE[29531] := 16#8AF8;
   // GBK_TO_UNICODE[29532] := 16#D655;
   // GBK_TO_UNICODE[29533] := 16#8AF9;
   // GBK_TO_UNICODE[29534] := 16#D656;
   // GBK_TO_UNICODE[29535] := 16#8AFA;
   // GBK_TO_UNICODE[29536] := 16#D657;
   // GBK_TO_UNICODE[29537] := 16#8AFB;
   // GBK_TO_UNICODE[29538] := 16#D658;
   // GBK_TO_UNICODE[29539] := 16#8AFC;
   // GBK_TO_UNICODE[29540] := 16#D659;
   // GBK_TO_UNICODE[29541] := 16#8AFD;
   // GBK_TO_UNICODE[29542] := 16#D65A;
   // GBK_TO_UNICODE[29543] := 16#8AFE;
   // GBK_TO_UNICODE[29544] := 16#D65B;
   // GBK_TO_UNICODE[29545] := 16#8AFF;
   // GBK_TO_UNICODE[29546] := 16#D65C;
   // GBK_TO_UNICODE[29547] := 16#8B00;
   // GBK_TO_UNICODE[29548] := 16#D65D;
   // GBK_TO_UNICODE[29549] := 16#8B01;
   // GBK_TO_UNICODE[29550] := 16#D65E;
   // GBK_TO_UNICODE[29551] := 16#8B02;
   // GBK_TO_UNICODE[29552] := 16#D65F;
   // GBK_TO_UNICODE[29553] := 16#8B03;
   // GBK_TO_UNICODE[29554] := 16#D660;
   // GBK_TO_UNICODE[29555] := 16#8B04;
   // GBK_TO_UNICODE[29556] := 16#D661;
   // GBK_TO_UNICODE[29557] := 16#8B05;
   // GBK_TO_UNICODE[29558] := 16#D662;
   // GBK_TO_UNICODE[29559] := 16#8B06;
   // GBK_TO_UNICODE[29560] := 16#D663;
   // GBK_TO_UNICODE[29561] := 16#8B08;
   // GBK_TO_UNICODE[29562] := 16#D664;
   // GBK_TO_UNICODE[29563] := 16#8B09;
   // GBK_TO_UNICODE[29564] := 16#D665;
   // GBK_TO_UNICODE[29565] := 16#8B0A;
   // GBK_TO_UNICODE[29566] := 16#D666;
   // GBK_TO_UNICODE[29567] := 16#8B0B;
